						);			
	WX4A_CP1_Out	:	CpABS_Out;
	WX4A_CP2_CI		: 	CpABS_CI := (
//						//bHomeStart_PI:= , 
//						//Stop_PI:= , 
//						//Reset_VI:= , 
//						//JogExecute_VI:= , 
//						//JogSlow_VI:= , 
//						//CW_VI:= , 
//						PPRset_CI:= 2 , 
//						cntPulseSet_CI:= 32778 , //set for 1 degree per pulse
//						HomingSet_CI:= 3 ,
//						GearRatio_CI:= 3 , 
//						Lead_CI:= 8 , 
//						MechDriveType_CI:= 2, 
//						InputFilter_CI:= 7 , 
//						SWLimit_Hi_CI:= 180 , 
//						SWLimit_Lo_CI:= -90, 
//						Limit_NC_NO_CI:= 1, 	//add sensor if more protection needed
//						ABSEncoderScaler_CI := 131,		//converts 1 cp pulse to encoder counts (scale and adjust this and cntPulseSet_CI to scale to imperial or metric)
//						ABSEncoderZero_CI := 2089769026 , //will need to change if 'cntPulseSet_CI' is changed or the tolerance will need to be checked to see how close to limit
//						ABSHiLimit_CI	:= 2089792841, //will need to change if 'cntPulseSet_CI' is changed or the tolerance will need to be checked to see how close to limit
//						ABSLoLimit_CI := 2089757112 //will need to change if 'cntPulseSet_CI' is changed or the tolerance will need to be checked to see how close to limit
//						//abs currently set for -90 deg to 180 deg
//						,
//						DisPerPulse_CI :=1,
//						MoveABSTol_CI :=1.5
						);			
	WX4A_CP2_Out	:	CpABS_Out;
	WX4A_CP3_CI		: 	CpABS_CI := (
//						//bHomeStart_PI:= , 
//						//Stop_PI:= , 
//						//Reset_VI:= , 
//						//JogExecute_VI:= , 
//						//JogSlow_VI:= , 
//						//CW_VI:= , 
//						PPRset_CI:= 2 , 
//						cntPulseSet_CI:= 800 , 
//						HomingSet_CI:= 2 ,
//						GearRatio_CI:= 3 , 
//						Lead_CI:= 8 , 
//						MechDriveType_CI:= 2, 
//						InputFilter_CI:= 7 , 
//						SWLimit_Hi_CI:= 100 , 
//						SWLimit_Lo_CI:= -125, 
//						Limit_NC_NO_CI:= 1,
//						DisPerPulse_CI :=1,
//						MoveABSTol_CI :=1.5
						
						);			
	WX4A_CP3_Out	:	CpABS_Out;
	WX4B_CP1_CI		: 	CpABS_CI := (
//						//bHomeStart_PI:= , 
//						//Stop_PI:= , 
//						//Reset_VI:= , 
//						//JogExecute_VI:= , 
//						//JogSlow_VI:= , 
//						//CW_VI:= , 
//						PPRset_CI:= 2 , 
//						cntPulseSet_CI:= 32000 , 
//						HomingSet_CI:= 3 ,
//						GearRatio_CI:= 3 , 
//						Lead_CI:= 8 , 
//						MechDriveType_CI:= 2, 
//						InputFilter_CI:= 7 , 
//						SWLimit_Hi_CI:= 150 , 
//						SWLimit_Lo_CI:= 0, 
//						Limit_NC_NO_CI:= 0, 
//						ABSEncoderScaler_CI := -950,		//converts 1 cp pulse to encoder counts (scale and adjust this and cntPulseSet_CI to scale to imperial or metric)
//						ABSEncoderZero_CI := 2117612704 , //will need to change if 'cntPulseSet_CI' is changed or the tolerance will need to be checked to see how close to limit
//						ABSHiLimit_CI	:= 2117613849, //will need to change if 'cntPulseSet_CI' is changed or the tolerance will need to be checked to see how close to limit
//						ABSLoLimit_CI := 2117469332 //will need to change if 'cntPulseSet_CI' is changed or the tolerance will need to be checked to see how close to limit
//						//swap ABS Hi and ABS Lo if encoder is mounted opposite.
//						,
//						DisPerPulse_CI :=1,
//						MoveABSTol_CI :=1.5
						);			
	WX4B_CP1_Out	:	CpABS_Out;
	WX4B_CP2_CI		: 	CpABS_CI := (
//						//bHomeStart_PI:= , 
//						//Stop_PI:= , 
//						//Reset_VI:= , 
//						//JogExecute_VI:= , 
//						//JogSlow_VI:= , 
//						//CW_VI:= , 
//						PPRset_CI:= 2 , 
//						cntPulseSet_CI:= 32778 , //set for 1 degree per pulse
//						HomingSet_CI:= 3 ,
//						GearRatio_CI:= 3 , 
//						Lead_CI:= 8 , 
//						MechDriveType_CI:= 2, 
//						InputFilter_CI:= 7 , 
//						SWLimit_Hi_CI:= 180 , 
//						SWLimit_Lo_CI:= -90, 
//						Limit_NC_NO_CI:= 1, 	//add sensor if more protection needed later
//						ABSEncoderScaler_CI := 132,		//converts 1 cp pulse to encoder counts (scale and adjust this and cntPulseSet_CI to scale to imperial or metric)
//						ABSEncoderZero_CI := 2117532059	 , //will need to change if 'cntPulseSet_CI' is changed or the tolerance will need to be checked to see how close to limit
//						ABSHiLimit_CI	:= 2117555547, //will need to change if 'cntPulseSet_CI' is changed or the tolerance will need to be checked to see how close to limit
//						ABSLoLimit_CI := 2117520354 //will need to change if 'cntPulseSet_CI' is changed or the tolerance will need to be checked to see how close to limit
//						//abs currently set for -90 deg to 180 deg
//						,
//						DisPerPulse_CI :=1,
//						MoveABSTol_CI :=1.5
						);
	WX4B_CP2_Out	:	CpABS_Out;
	
	WX4B_CP3_CI		: 	CpABS_CI := ( //not config yet
//						//bHomeStart_PI:= , 
//						//Stop_PI:= , 
//						//Reset_VI:= , 
//						//JogExecute_VI:= , 
//						//JogSlow_VI:= , 
//						//CW_VI:= , 
//						PPRset_CI:= 2 , 
//						cntPulseSet_CI:= 800 , 
//						HomingSet_CI:= 2 ,
//						GearRatio_CI:= 3 , 
//						Lead_CI:= 8 , 
//						MechDriveType_CI:= 2, 
//						InputFilter_CI:= 7 , 
//						SWLimit_Hi_CI:= 150 , 
//						SWLimit_Lo_CI:= 0, 
//						Limit_NC_NO_CI:= 1,
//						DisPerPulse_CI :=1,
//						MoveABSTol_CI :=1.5
						
						
						);			
	WX4B_CP3_Out	:	CpABS_Out;
						
END_VAR

// ---- Machine System/GVLs/GVL_Job.TcGVL
{attribute 'qualified_only'}
VAR_GLOBAL
	FinishedWithSprayZoneSD1 : BOOL;
	FinishedWithSprayZoneSD2 : BOOL;
	
END_VAR

// ---- Machine System/GVLs/GVL_Log.TcGVL
{attribute 'qualified_only'}
VAR_GLOBAL
	NewMeasure : BOOL;
	PointLogged : BOOL;
	ReadytoLog 	: BOOL := TRUE;
	
	XCur		: STRING;
	YCur		: STRING;
	ZCur		: STRING;
	RCur		: STRING;
	VCur		: STRING;
	Dist		: STRING;
	
	XRef		: STRING;
	YRef		: STRING;
	ZRef		: STRING;
	RRef		: STRING;
	VRef		: STRING;
	DistRef		: STRING;
	
	
END_VAR

// ---- Machine System/GVLs/GVL_SAF.TcGVL
{attribute 'qualified_only'}
VAR_GLOBAL
	Estop1a 		AT %Q* : BOOL;
	Estop1b 		AT %Q* : BOOL;
	ErrorAcknowledgment AT %Q* : BOOL;
	Run 			AT %Q* : BOOL;
	InRun			AT %I* : BOOL;
	ComErr			AT %I* : BOOL;
	FbErr			AT %I* : BOOL;
	EStopReset 		AT %Q* : BOOL;
	EStopMCR 		AT %I* : BOOL;
	EStopError 		AT %I* : BOOL;	//error from main estop safety fb block
	EStopError1		AT %I* : BOOL;	//error from c4 estop safety fb block (same safe inputs as main estop)
	EstopError2 	AT %I* : BOOL;	//error from c5 estop safety fb block (same safe inputs as main estop)
	WX_On 			AT %Q* : BOOL;	//plc variable to drive safety outputs for c4 and c5 contactors (wx boxes)
	EDM_Error_C4 	AT %I* : BOOL;
	EDM_Error_C5 	AT %I* : BOOL;
	EStopOK			AT %I* : BOOL;
	DeadmanEnable	AT %I* : BOOL;  //from C3:SI1
	
	//plc flag
	SafetyOk		AT %I* : BOOL;
END_VAR

// ---- Machine System/GVLs/GVL_IO.TcGVL
VAR_GLOBAL
	//Digital Inputs
	bEstopPB AT %I* : BOOL; 
	iFeedrateOverridePot AT %I* : INT := 32767;
	iSpindleOverridePot AT %I* : INT := 32767;
	iSpindleLoad AT %I* : INT;
	//home and limit sensors
	bXHomeSwitch AT %I* : BOOL;
	bYHomeSwitch AT %I* : BOOL;
	bZHomeSwitch AT %I* : BOOL;
	bAHomeSwitch AT %I* : BOOL;
	bCHomeSwitch AT %I* : BOOL;
	bHi_A AT %I* : BOOL;
	bLo_A AT %I* : BOOL;
	bHi_C AT %I* : BOOL;
	bLo_C AT %I* : BOOL;
	
	// Temperature Analog
	Thermocouple AT %I*: REAL := 0; // C3 EL3024 Channel 3 analog 4-20mA from thermocouple range 0-32767
	rAIInput1 : REAL;
	rAIInput2 : REAL;
	rAIInput3 : REAL;
	
	//Distance Analog
	iDistSens	AT %I*	: INT;	//analog distance sensor on z axis to measure tool
	
	//trunnion sensors
	bTrunCW AT %I* : BOOL;
	bTrunCCW AT %I* : BOOL;
	bTrun0 AT %I* : BOOL;
	bTrunOver AT %I* : BOOL;
	bTrunClampOn : BOOL :=true; // Trunnion clamp
	bTrunClampOnLast : BOOL :=TRUE; //Track state of clamp to disallow change while estop or enable off
	bTrunClampEn : BOOL;
	
	iTrunSig AT %Q*: INT;
	//Trunion Clearpath rotary
	//bEnable 	AT 	%Q* 	: BOOL;		//found in cprot function
	bEnableCom	AT 	%I* 	: BOOL;
	bAcom		AT	%I* 	: BOOL;
	//bAout		AT 	%Q*		: BOOL;		//found in cprot function
	bBcom		AT	%I* 	: BOOL;
	//bBout		AT 	%Q*		: BOOL;		//found in cprot function
	bHLFBcom	AT	%I* 	: BOOL;		//red wire
	bHLFB24V	AT 	%Q*		: BOOL; 	//green wire
	
	// gun valves
	bAceOn AT %Q* : BOOL;	// acetone gun mac valve
	bSprayOn AT %Q* : BOOL; // spray gun mac valve
	// smc valve outputs - one must be true and one must be false (a true b false or A false B true)
	bVa1A AT %Q* :BOOL;
	bVa1B AT %Q* :BOOL;
	bVa2A AT %Q* :BOOL;
	bVa2B AT %Q* :BOOL;
	bVa3A AT %Q* :BOOL;
	bVa3B AT %Q* :BOOL;
	bva4A AT %Q* : BOOL;
	bVa4B AT %Q* :BOOL;
	bVa5A AT %Q* :BOOL;
	bVa5B AT %Q* :BOOL;
	bVa6A AT %Q* :BOOL;
	bVa6B AT %Q* :BOOL;
	bVa7A AT %Q* :BOOL;
	bVa7B AT %Q* :BOOL;
	bVa8A AT %Q* :BOOL;
	bVa8B AT %Q* :BOOL;
	bVa9A AT %Q* :BOOL;
	bVa9B AT %Q* :BOOL;
	bVa10A AT %Q* :BOOL;
	bVa10B AT %Q* :BOOL;
	bVa11A AT %Q* :BOOL;
	bVa11B AT %Q* :BOOL;
	bVa12A AT %Q* :BOOL;
	bVa12B AT %Q* :BOOL;
	bVa13A AT %Q* :BOOL;	
	bVa13B AT %Q* :BOOL;
	bVa14A AT %Q* :BOOL;
	bVa14B AT %Q* :BOOL;
	bVa15A AT %Q* :BOOL;
	bVa15B AT %Q* :BOOL;
	bVa16A AT %Q* :BOOL;
	bVa16B AT %Q* :BOOL;
	
	WX1 : sBogie;
	WX2 : sBogie;
	WX3 : sBogie;
	WX4 : sBogie;
	
	//C6
	KM1_ContactorOn  AT %Q* : BOOL;
	KM2_ContactorOn  AT %Q* : BOOL;
	//C3
	FilterManometer AT %I*: INT; // Air Filter Elements differential pressure sensor
	gasSensor AT %I* : INT; // Styrene level sensor
	
END_VAR

// ---- Machine System/GVLs/GVL_Machine.TcGVL
VAR_GLOBAL
	pX: POINTER TO HIGH_LEVEL_INTERFACE_AX;
	pY: POINTER TO HIGH_LEVEL_INTERFACE_AX;
	pZ: POINTER TO HIGH_LEVEL_INTERFACE_AX;
	pCh0: POINTER TO HIGH_LEVEL_INTERFACE_CH;
	rX_ActPos : LREAL;
	rY_ActPos : LREAL;
	rZ_ActPos : LREAL;
	bAllAxisOkToEnable 	: BOOL;	
	bPLC_ForceEstop 	: BOOL;
	nCommandedRPM		: DINT;
	stVirtualHBA		: ARRAY[0..1] OF ST_CNCVirtualHBA;
	HeaterOnRequest		: LREAL;
	fSetpointValueToScope: LREAL;
	fActualValueToScope	 : LREAL;
	fOutToScope			: LREAL;
	fPIDLoop1ControlValue : LREAL;
	fPIDLoop1ProcessValue : LREAL;
	HeatOnRequest : BOOL;
	
END_VAR

VAR_GLOBAL CONSTANT
	MAX_CSV_ROWS 			: UDINT := 250;
	MAX_CSV_COLUMNS 		: UDINT := 1;
	MAX_CSV_FIELD_LENGTH	: UDINT := 100;
END_VAR

// ---- Machine System/PRGs/PID/PRG_PID_CALL.TcPOU
PROGRAM PRG_PID_CALL
VAR
	
END_VAR




// C3 EL3024 Channel 3 analog 4-20mA from thermocouple range 0-32767
// Measure -40F to 140F
GVL_IO.rAIInput3 := (Thermocouple/(32767.0 - 0.0))* 100;

HeaterOnRequest := PRG_FB_CTRL_PID.fOut;
PRG_FB_CTRL_PID();

//Call simulated PID for debugging locally. Comment out after commissioning
//PRG_SIM_PROCESS();

END_PROGRAM

// ---- Machine System/PRGs/PID/PRG_FB_CTRL_PID.TcPOU
PROGRAM PRG_FB_CTRL_PID
VAR
	fSetpointValue					: LREAL		:= 85.0;
	fActualValue					: LREAL;
	fManSyncValue					: LREAL;
	bSync							: BOOL;

	fOut							: LREAL;
	
	bHold							: BOOL;

	eMode							: E_CTRL_MODE;
	stCTRL_PID_PARAMS				: ST_CTRL_PID_PARAMS;

	eErrorId						: E_CTRL_ERRORCODES;
	bError							: BOOL;
	bARWactive						: BOOL;

	(* controller *)
	fbCTRL_PID						: FB_CTRL_PID;

	bInit							: BOOL	:= TRUE;
	fbTON							: TON;
	TcHmiToggleButtonHeaterOnOff    : BOOL;
END_VAR


	

IF bInit THEN
	(* init parameter struct *)
	stCTRL_PID_PARAMS.tCtrlCycleTime		:= T#500MS;
	stCTRL_PID_PARAMS.tTaskCycleTime		:= T#100MS;
	stCTRL_PID_PARAMS.fKp					:= 3.0;			(* proportional gain Kp				*)
	stCTRL_PID_PARAMS.tTn					:= T#20S;		(*  Tn								*)
	stCTRL_PID_PARAMS.tTv					:= T#200MS;		(*  Tv								*)
	stCTRL_PID_PARAMS.tTd					:= T#100MS;		(*  Td								*)
	stCTRL_PID_PARAMS.fOutMaxLimit			:=  100;		(* maximum output limit				*)
	stCTRL_PID_PARAMS.fOutMinLimit			:=  0.0;		(* minimum output limit				*)

	(* set the mode to ACTIVE --> normal operation *)
	eMode := eCTRL_MODE_ACTIVE;

	(* reset the init flag *)
	bInit := FALSE;
END_IF

(*TYPE E_CTRL_MODE :
(
    eCTRL_MODE_IDLE     := 0, 
    eCTRL_MODE_PASSIVE     := 1, 
    eCTRL_MODE_ACTIVE     := 2, 
    eCTRL_MODE_RESET     := 3, 
    eCTRL_MODE_MANUAL     := 4, 
    eCTRL_MODE_TUNE     := 5, 
    eCTRL_MODE_SELFTEST    := 6, 
    eCTRL_MODE_SYNC_MOVEMENT := 7 
)
END_TYPE*)

fActualValue := GVL_IO.rAIInput3; //Get process variable Temperature from analog input C3, AI1 Channel 3 value

(* copy var to scope var *)
GVL_Machine.fSetpointValueToScope 	:= fSetpointValue;
GVL_Machine.fActualValueToScope 	:= fActualValue;
GVL_Machine.fOutToScope 			:= fOut;

(* call controller *)
fbCTRL_PID(		fSetpointValue		:= fSetpointValue,
				fActualValue		:= fActualValue,
				fManSyncValue		:= fOut,
				bSync				:= bSync,
				eMode				:= eMode,
				bHold				:= bHold,
				stParams			:= stCTRL_PID_PARAMS,
				fOut				=> fOut,
				bARWactive			=> bARWactive,
				eErrorId			=> eErrorId,
				bError				=> bError
				);

(*IF eMode = 	eCTRL_MODE_ACTIVE THEN // Bumpless switch logic for switching PID for Manual to Automatic. The setpoint value needs TO follow the process value feedback
	fOut := fOut;		
END_IF				

IF eMode = 	eCTRL_MODE_ACTIVE THEN // Bumpless switch logic for switching PID for Automatic to Manual. The setpoint value needs to follow the process value feedback
	fSetpointValue := fActualValue;		
END_IF	*)

IF 	GVL_Machine.fOutToScope >= 10 OR TcHmiToggleButtonHeaterOnOff THEN
	 GVL_Machine.HeatOnRequest := TRUE;
	ELSE
	 GVL_Machine.HeatOnRequest := FALSE;
END_IF

END_PROGRAM

// ---- FAST.TcPOU
PROGRAM FAST
VAR
	nChan : INT;
	MOS_TS: INT;
END_VAR

(****************************************************************************************)
(*	  							Wait for HLI initialization								*)
(****************************************************************************************)
IF NOT CNCSystem.bHLIInit THEN
	RETURN;
END_IF

(* Programm call for MOS_TS M functions *)
// PRG_FastMFunctions();

END_PROGRAM

// ---- MAIN.TcPOU
PROGRAM MAIN
VAR
  
END_VAR



// everything related to time
	P_Timer();
	
	
// EventLogger
	P_EventLogger();

FirstScan();
// temporarily disabled by Kirk 
HLI3_Init(); 

//PRG_Sequence();
(* Call CNC related code only if the HLI has been initialized succesfully! *)
 IF CNCSystem.bHLIInit THEN
	PRG_CNCAxesHandler();    	
	PRG_CNCManualMode();
	PRG_CNCChannelHandler();	
	PRG_CNCVariablesViewer();
	PRG_ManualFnc();	
	myPRG_AxisHomeSwitches_1();
	myVE_Vars(); //call this before MCodes just to be sure data was pulled and updated for each potential MCODE Call [Add a buffer to mcode rtrig if ve does not compute from same gcode line call ie[ve.wxv=90 M510]
	myM_CODES();
////	myPressure();
//	myGun();
//	myCounter();
	mySafety();
	SafetyConnect();
	ModeHandle();
	//myHMIPLCRECIPE();
	//myDistance();
	WX_CP();
	WX_CP_Simple();
	Bogie();
	//myCNC_Call_Spray();
	CNC_HMI_HLI_Added_Code(); //display for new hmi variables
	BogieSettings();
	RollerDoors();
	PersonnelDoor();
	Heraus_Heater_Control();
	
//	 		(* Conveyor Programs *)
	
	Input_Buffering();
	MOTOR_FAULTS();
	JAM_FAULTS();
	OUTPUTS();
	//Ventilation();
	GL1_Transfer_Traverse();
	GL10_Transfer_Traverse();
	GL11_Transfer();
	GL2_Transfer();
	GL3_Accumulation();
	GL4_Accumulation();
	GL5A_Accumulation();
	GL5B_Accumulation();
	GL6_Conveyor();
	GL7_Conveyor();
	GL8_Conveyor();
	GL9_Conveyor();

			(* Rib Machine Programs *)
	Guarding_Safety();
	Input_Buffering_RB();
	START_STOP();
	Index_and_measure();
	Fault_Logic();
	Lift_Raise_and_Lower();
	Clamp_and_cut();
	Interlocks_to_Main_Line();
	// Outputs_RB();
	
END_IF
(* Reset the reset flag from HMI *)
PLCReset := FALSE;

END_PROGRAM

// ---- Machine System/PRGs/ALARM AND STATUS/P_Timer.TcPOU
PROGRAM P_Timer 
VAR
	fbSystemTime 		: FB_LocalSystemTime;
	dtCurrentDateTime 	: DT;
	sCurrentDateTime 	: STRING;
	sDateTime			: STRING;		
	bSecond				: BOOL;
	nSecond 			: WORD;
	bPulsels			: BOOL;
	
	fbRtSecond 			: R_TRIG;
	fbLow_ls			: TON;
	fbHigh_ls 			: TOF;
END_VAR

// synchronize system time 
	fbSystemTime(
		bEnable		:= TRUE, 
		dwCycle		:= 5, 
		dwOpt		:= 1
	);

	dtCurrentDateTime	:= SYSTEMTIME_TO_DT(fbSystemTime.systemTime); 
	sCurrentDateTime	:= MID(DT_TO_STRING(dtCurrentDateTime), 19, 4);

// convert timestamp because ':' invalid in file name 
	sDateTime := sCurrentDateTime; 
	sDateTime := replace (sDateTime,'-', 1, 11); 
	sDateTime := replace (sDateTime,'-', 1, 14); 
	sDateTime := replace (sDateTime,'-', 1, 17);
	
// 1 sec. trigger
	fbRtSecond (CLK 	:= fbSystemTime.systemTime.wSecond <> nSecond, Q => bSecond);
 	nSecond				:= fbSystemTime.systemTime.wSecond;
	
// 1 sec. blinking puls
	fbLow_ls(IN 		:= NOT bPulsels, PT:= T#500MS);
	fbHigh_ls(IN		:= fbLow_ls.Q,   PT:= T#500MS, Q => bPulsels);

END_PROGRAM

// ---- Machine System/PRGs/ALARM AND STATUS/P_EventLogger.TcPOU
PROGRAM P_EventLogger
VAR
	fbEventlogger		: FB_TcEventlogger;
	bClearAlarms		: BOOL;
	bConfirmAlarms 		: BOOL; 
	bClearLoggedEvents 	: BOOL; 
	bExportLoggedEvents : BOOL; 
	fbRtExport			: R_TRIG; 
	fbCsvExportSetting  : FB_TcEventCsvExportSettings; 
	fbExportFilter 		: FB_TcEventFilter; 
	sExportFileName 	: STRING := 'C:\temp\Eventlogger-export.csv';
	
	fbEventAlarm		: ARRAY[0..500] OF FB_EventAlarm;
	aClass1Alarm		: ARRAY[0..500] OF BOOL;	
	aClass2Alarm		: ARRAY[0..500] OF BOOL;	
	aClass3Alarm		: ARRAY[0..500] OF BOOL;	
	fbEventWarning 		: ARRAY[0..500] OF FB_EventMessage;
	aWarning			: ARRAY[0..512] OF BOOL;
	fbEventInfo 		: ARRAY[0..500] OF FB_EventMessage;
	aInfo				: ARRAY[0..500] OF BOOL;
  
	hr					: HRESULT;
	hrLastError 		: HRESULT;
	
END_VAR

Event_Calls(); 				// Program to turn Alarms on
a_010_AlarmsClass1(); 		// alarms class 1, emergency stop, safety doors, power supply, etc.
a_010_AlarmsClass2(); 		// alarms class 2, movements, drives, pneumatic cylinder, etc.
a_010_AlarmsClass3(); 		// alarms class 3, process, level, temperature, conductivity, etc.

a_020_Warnings(); 			// warnings, filter change, refilling of tanks, pre-alarms, etc.

a_030_Infos(); 				// messages, audit-trail, etc.

a_040_ConfirmLoggedAlarms();// confirm all logged alarms

(*a_050_ClearLoggedAlarms ();// clear all logged events PLC*)

a_060_ClearLoggedEvents(); // clear all logged events PLC

a_070_ExportLoggedEvents();// export logged events csv file

ACTION a_010_AlarmsClass1:

//Alarms Class 1 
	fbEventAlarm[0](
		bEvent			:=	aClass1Alarm[0],
		nEventID		:=	4096,
		sSource			:=	'TwinSAFE Program'
	);
	fbEventAlarm[1](
		bEvent			:=	aClass1Alarm[1],
		nEventID		:=	4097,
		sSource			:=	'GL1 Motor Fault'
	);
	fbEventAlarm[2](
		bEvent			:=	aClass1Alarm[2],
		nEventID		:=	4098,
		sSource			:=	'GL2 Motor Fault'
	);
	fbEventAlarm[3](
		bEvent			:=	aClass1Alarm[3],
		nEventID		:=	4099,
		sSource			:=	'GL3 Motor Fault'
	);
	fbEventAlarm[4](
		bEvent			:=	aClass1Alarm[4],
		nEventID		:=	4100,
		sSource			:=	'GL4 Motor Fault'
	);
	fbEventAlarm[5](
		bEvent			:=	aClass1Alarm[5],
		nEventID		:=	4101,
		sSource			:=	'GL5A Motor Fault'
	);
	fbEventAlarm[6](
		bEvent			:=	aClass1Alarm[6],
		nEventID		:=	4102,
		sSource			:=	'GL5B Motor Fault'
	);
	fbEventAlarm[7](
		bEvent			:=	aClass1Alarm[7],
		nEventID		:=	4103,
		sSource			:=	'GL6 Motor Fault'
	);
	fbEventAlarm[8](
		bEvent			:=	aClass1Alarm[8],
		nEventID		:=	4104,
		sSource			:=	'GL7 Motor Fault'
	);
	fbEventAlarm[9](
		bEvent			:=	aClass1Alarm[9],
		nEventID		:=	4105,
		sSource			:=	'GL8 Motor Fault'
	);
	fbEventAlarm[10](
		bEvent			:=	aClass1Alarm[10],
		nEventID		:=	4106,
		sSource			:=	'GL9 Motor Fault'
	);
	fbEventAlarm[11](
		bEvent			:=	aClass1Alarm[11],
		nEventID		:=	4107,
		sSource			:=	'GL10 Motor Fault'
	);
	fbEventAlarm[12](
		bEvent			:=	aClass1Alarm[12],
		nEventID		:=	4108,
		sSource			:=	'GL11 Motor Fault'
	);
	fbEventAlarm[13](
		bEvent			:=	aClass1Alarm[13],
		nEventID		:=	4109,
		sSource			:=	'GL12 Motor Fault'
	);
END_ACTION

ACTION a_010_AlarmsClass2:
//Alarms Class 2 
	fbEventAlarm[14](
		bEvent			:=	aClass2Alarm[0],
		nEventID		:=	8192,
		sSource			:=	'GL1 jam'
	);
	fbEventAlarm[15](
		bEvent			:=	aClass2Alarm[1],
		nEventID		:=	8193,
		sSource			:=	'GL2 jam'
	);
	fbEventAlarm[16](
		bEvent			:=	aClass2Alarm[2],
		nEventID		:=	8194,
		sSource			:=	'GL3 jam'
	);
	fbEventAlarm[17](
		bEvent			:=	aClass2Alarm[3],
		nEventID		:=	8195,
		sSource			:=	'GL4 jam'
	);
	fbEventAlarm[18](
		bEvent			:=	aClass2Alarm[4],
		nEventID		:=	8196,
		sSource			:=	'GL5A jam'
	);
	fbEventAlarm[19](
		bEvent			:=	aClass2Alarm[5],
		nEventID		:=	8197,
		sSource			:=	'GL5B jam'
	);
	fbEventAlarm[20](
		bEvent			:=	aClass2Alarm[6],
		nEventID		:=	8198,
		sSource			:=	'GL6 jam'
	);
	fbEventAlarm[21](
		bEvent			:=	aClass2Alarm[7],
		nEventID		:=	8199,
		sSource			:=	'GL7 jam'
	);
	fbEventAlarm[22](
		bEvent			:=	aClass2Alarm[8],
		nEventID		:=	8200,
		sSource			:=	'GL8 jam'
	);
	fbEventAlarm[23](
		bEvent			:=	aClass2Alarm[9],
		nEventID		:=	8201,
		sSource			:=	'GL9 jam'
	);
	fbEventAlarm[24](
		bEvent			:=	aClass2Alarm[10],
		nEventID		:=	8202,
		sSource			:=	'GL10 jam'
	);
	fbEventAlarm[25](
		bEvent			:=	aClass2Alarm[11],
		nEventID		:=	8203,
		sSource			:=	'GL11 jam'
	);
	fbEventAlarm[26](
		bEvent			:=	aClass2Alarm[12],
		nEventID		:=	8204,
		sSource			:=	'GL12 jam'
	);
END_ACTION

ACTION a_010_AlarmsClass3:
//Alarms Class 3 
	fbEventAlarm[30](
		bEvent			:=	aClass3Alarm[0],
		nEventID		:=	4116,
		sSource			:=	'Air Filter'
	);
	fbEventAlarm[31](
		bEvent			:=	aClass3Alarm[1],
		nEventID		:=	4117,
		sSource			:=	'Air Filter'
	);
	fbEventAlarm[32](
		bEvent			:=	aClass3Alarm[2],
		nEventID		:=	4118,
		sSource			:=	'Styrene'
	);
	fbEventAlarm[33](
		bEvent			:=	aClass3Alarm[3],
		nEventID		:=	4119,
		sSource			:=	'Class3Alarm 3'
	);
	fbEventAlarm[34](
		bEvent			:=	aClass3Alarm[4],
		nEventID		:=	4120,
		sSource			:=	'Class3Alarm 4'
	);
	fbEventAlarm[35](
		bEvent			:=	aClass3Alarm[5],
		nEventID		:=	4121,
		sSource			:=	'Class3Alarm 5'
	);
	fbEventAlarm[36](
		bEvent			:=	aClass3Alarm[6],
		nEventID		:=	4122,
		sSource			:=	'Class3Alarm 6'
	);
	fbEventAlarm[37](
		bEvent			:=	aClass3Alarm[7],
		nEventID		:=	4123,
		sSource			:=	'Class3Alarm 7'
	);
	fbEventAlarm[38](
		bEvent			:=	aClass3Alarm[8],
		nEventID		:=	4124,
		sSource			:=	'Class3Alarm 8'
	);
	fbEventAlarm[39](
		bEvent			:=	aClass3Alarm[9],
		nEventID		:=	4125,
		sSource			:=	'Class3Alarm 9'
	);
END_ACTION

ACTION a_020_Warnings:
// Warning 
	fbEventWarning[0](
		bEvent 		:= 	aWarning[0],
		nEventID	:=	1280,
		sSource		:=	'Styrene Level'
	);
	fbEventWarning[1](
		bEvent 		:= 	aWarning[1],
		nEventID	:=	1281,
		sSource		:=	'Roll Door 1'
	);
	fbEventWarning[2](
		bEvent 		:= 	aWarning[2],
		nEventID	:=	1282,
		sSource		:=	'Roll Door 2'
	);
	fbEventWarning[3](
		bEvent 		:= 	aWarning[3],
		nEventID	:=	1283,
		sSource		:=	'Roll Door 3'
	);
	fbEventWarning[4](
		bEvent 		:= 	aWarning[4],
		nEventID	:=	1284,
		sSource		:=	'Warning 4'
	);
	fbEventWarning[5](
		bEvent 		:= 	aWarning[5],
		nEventID	:=	1285,
		sSource		:=	'Warning 5'
	);
	fbEventWarning[6](
		bEvent 		:= 	aWarning[6],
		nEventID	:=	1286,
		sSource		:=	'Warning 6'
	);
	fbEventWarning[7](
		bEvent 		:= 	aWarning[7],
		nEventID	:=	1287,
		sSource		:=	'Warning 7'
	);
	fbEventWarning[8](
		bEvent 		:= 	aWarning[8],
		nEventID	:=	1288,
		sSource		:=	'Warning 8'
	);
	fbEventWarning[9](
		bEvent 		:= 	aWarning[9],
		nEventID	:=	1289,
		sSource		:=	'Warning 9'
	);
	fbEventWarning[10](
		bEvent 		:= 	aWarning[10],
		nEventID	:=	1290,
		sSource		:=	'Warning 10'
	);
	fbEventWarning[11](
		bEvent 		:= 	aWarning[11],
		nEventID	:=	1291,
		sSource		:=	'Warning 11'
	);
	fbEventWarning[12](
		bEvent 		:= 	aWarning[12],
		nEventID	:=	1292,
		sSource		:=	'Warning 12'
	);
	fbEventWarning[13](
		bEvent 		:= 	aWarning[13],
		nEventID	:=	1293,
		sSource		:=	'Warning 13'
	);
	fbEventWarning[14](
		bEvent 		:= 	aWarning[14],
		nEventID	:=	1294,
		sSource		:=	'Warning 14'
	);
	fbEventWarning[15](
		bEvent 		:= 	aWarning[15],
		nEventID	:=	1295,
		sSource		:=	'Warning 15'
	);
	fbEventWarning[16](
		bEvent 		:= 	aWarning[16],
		nEventID	:=	1296,
		sSource		:=	'Warning 16'
	);
	fbEventWarning[17](
		bEvent 		:= 	aWarning[17],
		nEventID	:=	1297,
		sSource		:=	'Warning 17'
	);
	fbEventWarning[18](
		bEvent 		:= 	aWarning[18],
		nEventID	:=	1298,
		sSource		:=	'Warning 18'
	);
	fbEventWarning[19](
		bEvent 		:= 	aWarning[19],
		nEventID	:=	1299,
		sSource		:=	'Warning 19'
	);
END_ACTION

ACTION a_030_Infos:
// Info 
	fbEventInfo[0](
		bEvent 		:= 	aInfo[0],
		nEventID	:=	0,
		sSource		:=	'Info 0'
	);
	fbEventInfo[1](
		bEvent 		:= 	aInfo[1],
		nEventID	:=	1,
		sSource		:=	'Info 1'
	);
	fbEventInfo[2](
		bEvent 		:= 	aInfo[2],
		nEventID	:=	2,
		sSource		:=	'Info 2'
	);
	fbEventInfo[3](
		bEvent 		:= 	aInfo[3],
		nEventID	:=	3,
		sSource		:=	'Info 3'
	);
	fbEventInfo[4](
		bEvent 		:= 	aInfo[4],
		nEventID	:=	4,
		sSource		:=	'Info 4'
	);
	fbEventInfo[5](
		bEvent 		:= 	aInfo[5],
		nEventID	:=	5,
		sSource		:=	'Info 5'
	);
	fbEventInfo[6](
		bEvent 		:= 	aInfo[6],
		nEventID	:=	6,
		sSource		:=	'Info 6'
	);
	fbEventInfo[7](
		bEvent 		:= 	aInfo[7],
		nEventID	:=	7,
		sSource		:=	'Info 7'
	);
	fbEventInfo[8](
		bEvent 		:= 	aInfo[8],
		nEventID	:=	8,
		sSource		:=	'Info 8'
	);
	fbEventInfo[9](
		bEvent 		:= 	aInfo[9],
		nEventID	:=	9,
		sSource		:=	'Info 9'
	);
	fbEventInfo[10](
		bEvent 		:= 	aInfo[10],
		nEventID	:=	10,
		sSource		:=	'Info 10'
	);
	fbEventInfo[11](
		bEvent 		:= 	aInfo[11],
		nEventID	:=	11,
		sSource		:=	'Info 11'
	);
	fbEventInfo[12](
		bEvent 		:= 	aInfo[12],
		nEventID	:=	12,
		sSource		:=	'Info 12'
	);
	fbEventInfo[13](
		bEvent 		:= 	aInfo[13],
		nEventID	:=	13,
		sSource		:=	'Info 13'
	);
	fbEventInfo[14](
		bEvent 		:= 	aInfo[14],
		nEventID	:=	14,
		sSource		:=	'Info 14'
	);
	fbEventInfo[15](
		bEvent 		:= 	aInfo[15],
		nEventID	:=	15,
		sSource		:=	'Info 15'
	);
	fbEventInfo[16](
		bEvent 		:= 	aInfo[16],
		nEventID	:=	16,
		sSource		:=	'Info 16'
	);
	fbEventInfo[17](
		bEvent 		:= 	aInfo[17],
		nEventID	:=	17,
		sSource		:=	'Info 17'
	);
	fbEventInfo[18](
		bEvent 		:= 	aInfo[18],
		nEventID	:=	18,
		sSource		:=	'Info 18'
	);
	fbEventInfo[19](
		bEvent 		:= 	aInfo[19],
		nEventID	:=	19,
		sSource		:=	'Info 19'
	);
END_ACTION

ACTION a_040_ConfirmLoggedAlarms:
// confirmation of all alarms	

	IF bConfirmAlarms THEN
			hr:= fbEventLogger.ConfirmAllAlarms(0);
			IF FAILED(hr) THEN
				hrLastError := hr;
			END_IF
	END_IF
END_ACTION

ACTION a_050_ClearLoggedAlarms:
// reset ALL Alarms 
// must not be used!!! I reset the alarms in the corresponding instances

	(*IF bClearAlarms THEN
			hr := fbEventlogger.ClearAllAlarms(0,FALSE);
			IF FAILED(hr) THEN
					hrLastError := hr;
			END_IF
	END_IF*)
END_ACTION

ACTION a_060_ClearLoggedEvents:
// clear all logged events PLC Cache
	IF bClearLoggedEvents THEN
		bClearLoggedEvents := FALSE;
		fbEventlogger.ClearLoggedEvents(0);
	END_IF
END_ACTION

ACTION a_070_ExportLoggedEvents:
// create file name
	sExportFileName := CONCAT(CONCAT('C:\Temp\',P_Timer.sDateTime), '.csv');
	
// CSV export logged events. Without filter all logged events will be exported. 
// CSV file will be overvritten, an opened file fires an error
	fbRtExport (CLK:= bExportLoggedEvents); 
	IF bExportLoggedEvents THEN 
		IF fbRtExport.Q THEN
			fbCsvExportSetting.Clear(); 
			fbCsvExportSetting.AddLanguage(1031, 'German'); 
		//	fbCsvExportSetting. AddFilter (fbExportFilter);
		//	fbExportFilter.Clear().IsAlarm()AND_OP().EventClass.EqualTO (TC_EVENTS.myAlarmEventClass.x1000.uuidEventClass); 
		END_IF 
		IF fbEventLogger.ExportLoggedEvents(sExportFileName,fbCsvExportSetting, hrErrorCode=> hr) THEN
			bExportLoggedEvents:= FALSE; 
		END_IF 
	END_IF
END_ACTION

ACTION Event_Calls:


// alarms class 1, emergency stop, safety doors, power supply, etc.
	IF NOT gvl_saf.SafetyOk THEN aClass1Alarm[0] := 1; ELSE aClass1Alarm[0] := 0; END_IF
		
/////////////////////////// CONVEYOR MOTOR FAULTS
	
	
	IF GVL_Conveyors.GL1.Motor_Fault THEN aClass1Alarm[1] := 1; ELSE aClass1Alarm[1] := 0; END_IF // GL1 MOTOR FAULT
	
	IF GVL_Conveyors.GL2.Motor_Fault THEN aClass1Alarm[2] := 1; ELSE aClass1Alarm[2] := 0; END_IF // GL2 MOTOR FAULT
		
	IF GVL_Conveyors.GL3.Motor_Fault THEN aClass1Alarm[3] := 1; ELSE aClass1Alarm[3] := 0; END_IF // GL3 MOTOR FAULT
	
	IF GVL_Conveyors.GL4.Motor_Fault THEN aClass1Alarm[4] := 1; ELSE aClass1Alarm[4] := 0; END_IF // GL4 MOTOR FAULT
	
	IF GVL_Conveyors.GL5A.Motor_Fault THEN aClass1Alarm[5] := 1; ELSE aClass1Alarm[5] := 0; END_IF // GL5A MOTOR FAULT
	
	IF GVL_Conveyors.GL5B.Motor_Fault THEN aClass1Alarm[6] := 1; ELSE aClass1Alarm[5] := 0; END_IF // GL5B MOTOR FAULT
		
	IF GVL_Conveyors.GL6.Motor_Fault THEN aClass1Alarm[7] := 1; ELSE aClass1Alarm[7] := 0; END_IF // GL6 MOTOR FAULT
	
	IF GVL_Conveyors.GL7.Motor_Fault THEN aClass1Alarm[8] := 1; ELSE aClass1Alarm[8] := 0; END_IF // GL7 MOTOR FAULT
	
	IF GVL_Conveyors.GL8.Motor_Fault THEN aClass1Alarm[9] := 1; ELSE aClass1Alarm[9] := 0; END_IF // GL8 MOTOR FAULT
	
	IF GVL_Conveyors.GL9.Motor_Fault THEN aClass1Alarm[10] := 1; ELSE aClass1Alarm[10] := 0; END_IF // GL9 MOTOR FAULT
		
	IF GVL_Conveyors.GL10.Motor_Fault THEN aClass1Alarm[11] := 1; ELSE aClass1Alarm[11] := 0; END_IF // GL10 MOTOR FAULT
	
	IF GVL_Conveyors.GL11.Motor_Fault THEN aClass1Alarm[12] := 1; ELSE aClass1Alarm[12] := 0; END_IF // GL11 MOTOR FAULT
	
	IF GVL_Conveyors.GL12.Motor_Fault THEN aClass1Alarm[13] := 1; ELSE aClass1Alarm[13] := 0; END_IF // GL12 MOTOR FAULT
	
	
	//////////////////////////////CONVEYOR JAM FAULTS
	// alarms class 2, movements, drives, pneumatic cylinder, etc.
	
	IF GVL_Conveyors.GL1.Jam_Fault 	THEN aClass2Alarm[0] := 1; ELSE aClass2Alarm[0] := 0; END_IF // GL1 JAM FAULT
		
	IF GVL_Conveyors.GL2.Jam_Fault 	THEN aClass2Alarm[1] := 1; ELSE aClass2Alarm[1] := 0; END_IF // GL2 JAM FAULT
	
	IF GVL_Conveyors.GL3.Jam_Fault 	THEN aClass2Alarm[2] := 1; ELSE aClass2Alarm[2] := 0; END_IF // GL3 JAM FAULT
	
	IF GVL_Conveyors.GL4.Jam_Fault 	THEN aClass2Alarm[3] := 1; ELSE aClass2Alarm[3] := 0; END_IF // GL4 JAM FAULT
	
	IF GVL_Conveyors.GL5A.Jam_Fault	THEN aClass2Alarm[4] := 1; ELSE aClass2Alarm[4] := 0; END_IF // GL5A JAM FAULT

	IF GVL_Conveyors.GL5B.Jam_Fault	THEN aClass2Alarm[5] := 1; ELSE aClass2Alarm[5] := 0; END_IF // GL5B JAM FAULT
		
	IF GVL_Conveyors.GL6.Jam_Fault	THEN aClass2Alarm[6] := 1; ELSE aClass2Alarm[6] := 0; END_IF // GL6 JAM FAULT

	IF GVL_Conveyors.GL7.Jam_Fault	THEN aClass2Alarm[7] := 1; ELSE aClass2Alarm[7] := 0; END_IF // GL7 JAM FAULT
		
	IF GVL_Conveyors.GL8.Jam_Fault	THEN aClass2Alarm[8] := 1; ELSE aClass2Alarm[8] := 0; END_IF // GL8 JAM FAULT
		
	IF GVL_Conveyors.GL9.Jam_Fault	THEN aClass2Alarm[9] := 1; ELSE aClass2Alarm[9] := 0; END_IF // GL9 JAM FAULT
	
	IF GVL_Conveyors.GL10.Jam_Fault	THEN aClass2Alarm[10] := 1; ELSE aClass2Alarm[10] := 0; END_IF // GL10 JAM FAULT
		
	IF GVL_Conveyors.GL11.Jam_Fault	THEN aClass2Alarm[11] := 1; ELSE aClass2Alarm[11] := 0; END_IF // GL11 JAM FAULT
	
	IF GVL_Conveyors.GL12.Jam_Fault	THEN aClass2Alarm[12] := 1; ELSE aClass2Alarm[12] := 0; END_IF // GL12 JAM FAULT
	
	

// alarms class 3, process, level, temperature, conductivity, etc.

	IF Ventilation.FILTER_CHANGE_NEEDED		THEN aClass3Alarm[0] := 1; ELSE aClass3Alarm[0] := 0; END_IF
	
	IF Ventilation.FILTER_OBSTRUCTED_FAULT THEN aClass3Alarm[1] := 1; ELSE aClass3Alarm[1] := 0; END_IF
		
	IF Ventilation.gasSensorFaulted		THEN aClass3Alarm[2] := 1; ELSE aClass3Alarm[2] := 0; END_IF
	
		
	//IF NewBatch.ResinTote.ActualScaleWeight < NewBatch.ResinTote.EmptyScaleWeight
	//									THEN aClass3Alarm[2] := 1; ELSE aClass3Alarm[2] := 0; END_IF
		
	//IF GVL.FiltersNeedChangeOutMain		THEN aClass3Alarm[3] := 1; ELSE aClass3Alarm[3] := 0; END_IF
		
	//IF GVL.FiltersNeedChangeOutSpecial	THEN aClass3Alarm[4] := 1; ELSE aClass3Alarm[4] := 0; END_IF
		
	//IF NewBatch.MixerCaseStep = 900		THEN aClass3Alarm[5] := 1; ELSE aClass3Alarm[5] := 0; END_IF
		
	//IF NewBatch.HoldTank.ActualScaleWeight > NewBatch.HoldTank.FullScaleWeight   						
	//									THEN aClass3Alarm[6] := 1; ELSE aClass3Alarm[6] := 0; END_IF
	
		
// warnings, filter change, refilling of tanks, pre-alarms, etc.

	//IF Ventilation.FILTER_OBSTRUCTED_FAULT	THEN aWarning[0] := 1; ELSE aWarning[0] := 0; END_IF
		
	//IF HMI.Filter2.ChangeOutNeededAlarm = 1		THEN aWarning[1] := 1; ELSE aWarning[1] := 0; END_IF
		
	//IF HMI.Filter3.ChangeOutNeededAlarm = 1		THEN aWarning[2] := 1; ELSE aWarning[2] := 0; END_IF
		
	//IF HMI.Filter4.ChangeOutNeededAlarm = 1		THEN aWarning[3] := 1; ELSE aWarning[3] := 0; END_IF
		
	//IF NewBatch.IngredientsReady = 0			THEN aWarning[4] := 1; ELSE aWarning[4] := 0; END_IF
		
	
// Infos

	IF GVL_Conveyors.ALL_CONVEYORS_IN_CYCLE AND  GVL_CONVEYORS.MOTOR_FAULT_WORD = 0 AND GVL_CONVEYORS.JAM_FAULT_WORD =0 THEN aInfo[0] := 1; ELSE aInfo[0] := 0; END_IF
		
	IF NOT GVL_Conveyors.ALL_CONVEYORS_IN_CYCLE AND  GVL_CONVEYORS.MOTOR_FAULT_WORD = 0 AND GVL_CONVEYORS.JAM_FAULT_WORD =0 THEN aInfo[1] := 1; ELSE aInfo[1] := 0; END_IF
		
	//IF HMI.Filter2.ChangeOutCompleted THEN aInfo[1] := 1; ELSE aInfo[1] := 0; END_IF
END_ACTION

END_PROGRAM

// ---- Machine System/FBs/EventLogger/FB_EventAlarm.TcPOU
FUNCTION_BLOCK FB_EventAlarm
VAR_INPUT 
	bEvent			: BOOL; 
	nEventID		: UDINT; 
	sSource			: STRING; 
END_VAR 
VAR_OUTPUT 
END_VAR
VAR 
	bIsInitalized	: BOOL;
	
	fbSourceInfo 	: FB_TcSourceInfo;
	fbAlarm 		: FB_TCAlarm;
	eventEntry 		: TcEventEntry;
	fbRtEvent 		: R_TRIG;
	fbFtEvent		: F_TRIG;
	
	hr				: HRESULT; 
	hrLastError 	: HRESULT;
	
END_VAR

// Initialization 
	IF NOT bIsInitalized THEN
		bIsInitalized:= TRUE;
		
		eventEntry:= Tc_Events.myAlarmEventClass.x1000; 
		eventEntry.nEventId:= nEventID;
		
		fbSourceInfo.Clear(); 
		fbSourceInfo.sName:= sSource;
		
		hr:= fbAlarm.CreateEx(eventEntry, TRUE, ipSourceInfo:= fbSourceInfo); 
		IF FAILED(hr) THEN
			hrLastError:= hr; 
		END_IF 
	END_IF
	
// event trigger 
	fbRtEvent(CLK:= bEvent); 
	fbFtEvent (CLK:= bEvent);
	
// alarm raised 
	IF  fbRtEvent.Q THEN
		hr:= fbAlarm.Raise(0); 
		IF FAILED(hr) THEN
			hrLastError:= hr; 
		END_IF
	END_IF
	
// alarm cleared 
	IF fbFtEvent.Q THEN
		hr:= fbAlarm.Clear(0, bResetConfirmation:= TRUE); 
		IF FAILED(hr) THEN
			hrLastError:= hr; 
		END_IF 
	END_IF

END_FUNCTION_BLOCK

// ---- Machine System/FBs/EventLogger/FB_EventMessage.TcPOU
FUNCTION_BLOCK FB_EventMessage 
VAR_INPUT 
	bEvent			: BOOL; 
	nEventID		: UDINT; 
	sSource			: STRING; 
END_VAR 
VAR_OUTPUT 
END_VAR 
VAR
	bIsInitalized : BOOL;
	
	fbSourceInfo 	: FB_TcSourceInfo;
	fbMessage 		: FB_TcMessage;
	eventEntry 		: TcEventEntry;
	fbRtEvent		: R_TRIG;
	hr 				: HRESULT;
	hrLastError		: HRESULT;
	
END_VAR

// initialization 
	IF NOT bIsInitalized THEN
		bIsInitalized:= TRUE;
		
		IF nEventID> 16#04FF THEN
			eventEntry:= Tc_Events.myWarningEventClass.x0500; 
		ELSE
			eventEntry:= TC_Events.myInfoEventClass.x0000; 
		END_IF
		
		eventEntry.nEventId:= nEventID;
		fbSourceInfo.Clear(); 
		fbSourceInfo.sName := sSource;
		
		hr:= fbMessage.CreateEx(eventEntry, ipSourceInfo:= fbSourceInfo); 
		IF FAILED (hr) THEN
			hrLastError:= hr; 
		END_IF 
	END_IF
	
// event trigger 
	fbRtEvent (CLK:= bEvent);

// message sent
	IF fbRtEvent.Q THEN
		hr:= fbMessage. Send(0); 
		IF FAILED (hr) THEN
			hrLastError:= hr;
		END_IF 
	END_IF

END_FUNCTION_BLOCK

// ---- Machine System/PRGs/Ventilation.TcPOU
PROGRAM Ventilation
VAR_INPUT
	SettingsArray :  ARRAY[1..2] OF sDatagridVFD;
END_VAR
VAR
	
	VentAreaRequest : BOOL;
	VentAreaTimer 	: TON;
	
	TrenchFanMtr : sVFD;
	FilterBankFanMtr : sVFD;
	
	
	gasSensorNormal  : BOOL;
	gasSensorHigh  : BOOL;
	gasSensorFaulted  : BOOL;
	

	FILTER_CHANGE_NEEDED : BOOL;
	FILTER_OBSTRUCTED_FAULT : BOOL;
	FILTER_OK : BOOL;

	filterCheck : UINT;
	StyreneCheck : UINT;
	ScaledManometer : REAL;
	ScaledStyrene : REAL;
	Results: real;
END_VAR


//setting of the ID strings for the settings page
SettingsArray[1].NameVFD := 'Filter Bank';
SettingsArray[2].NameVFD := 'Trench';

//outputing speed to settings page
SettingsArray[1].CurrentSpeed := FilterBankFanMtr.CurrentSpeed;
SettingsArray[2].CurrentSpeed := TrenchFanMtr.CurrentSpeed;


// Run Vfd Controlled Vent Fans At Optimal Speed Unless Gas Sensor Reads High
IF NOT gasSensorNormal THEN 
	TrenchFanMtr.RunRequest 	:= 1; 
	FilterBankFanMtr.RunRequest := 1; 
    TrenchFanMtr.SpeedRequested 	:= SettingsArray[2].SpeedSetpointLow;
	FilterBankFanMtr.SpeedRequested := SettingsArray[1].SpeedSetpointLow;
	ELSE
	TrenchFanMtr.RunRequest 	:= 1; 
	FilterBankFanMtr.RunRequest := 1; 
    TrenchFanMtr.SpeedRequested 	:= SettingsArray[2].SpeedSetpointHigh;
	FilterBankFanMtr.SpeedRequested := SettingsArray[1].SpeedSetpointHigh;
END_IF


// Manometer for air filters. Analog scaled to 0-100
						
ScaledManometer := ((INT_TO_REAL(GVL_IO.FilterManometer) / 32767 - 0.0)* 100); //* 20; // SCALE OF ANALOG INPUT 0-100

IF ScaledManometer <  49 THEN // ScaledManomter is scaled value from Manometer 0-100. Check that its not to halfway of full range yet.
	filterCheck := 1;
END_IF

IF ScaledManometer >  50 AND ScaledManometer < 80 THEN // ScaledManometer is scaled value from Manometer 0-100. Check if its over halfway of full range yet.
	filterCheck := 2;
END_IF

IF ScaledManometer >  80 OR ScaledManometer < 0 THEN // ScaledManometer is scaled value from Manometer 0-100. Check if its over 80% of full range yet.
	filterCheck := 3;
END_IF
	

CASE filterCheck OF 
     1 : FILTER_OK := TRUE; 
         FILTER_CHANGE_NEEDED := FALSE;
		 FILTER_OBSTRUCTED_FAULT := FALSE; 

     2 : FILTER_CHANGE_NEEDED := TRUE; 
         FILTER_OK := FALSE; 
		 FILTER_OBSTRUCTED_FAULT := FALSE;

	 3 : FILTER_OK := FALSE; 
         FILTER_OBSTRUCTED_FAULT:= TRUE;
		 FILTER_CHANGE_NEEDED := FALSE;
ELSE 
	 FILTER_OK := FALSE;
	 FILTER_OBSTRUCTED_FAULT := FALSE;
	 FILTER_CHANGE_NEEDED := FALSE;
END_CASE;


// Styrene Gas Sensor. Analog scaled to 0-100
//gasSensor := 16000;				
ScaledStyrene := ((INT_TO_REAL(GVL_IO.GasSensor) / 32767 - 0.0)* 100); // SCALE OF ANALOG INPUT 0-100

IF ScaledStyrene <  49 THEN // ScaledStyrene is scaled value from Styrene gas sensor 0-100.  Check that its not to halfway of full range yet.
	StyreneCheck := 1;
END_IF

IF ScaledStyrene >  50 AND ScaledStyrene < 80 THEN // ScaledStyrene is scaled value from Styrene gas sensor 0-100.  Check if its over halfway of full range yet.
	StyreneCheck := 2;
END_IF

IF ScaledStyrene >  80 OR ScaledStyrene < 0 THEN // ScaledStyrene is scaled value from Styrene gas sensor 0-100. Check if its over 80% of full range yet.
	StyreneCheck := 3;
END_IF
	

CASE StyreneCheck OF 
     1 : gasSensorNormal := TRUE; 
         gasSensorHigh := FALSE;
		 gasSensorFaulted := FALSE; 

     2 : gasSensorNormal := FALSE; 
	 	 gasSensorHigh := TRUE;
		 gasSensorFaulted := FALSE;

	 3 : gasSensorNormal := FALSE; 
         gasSensorHigh := FALSE;
		 gasSensorFaulted:= TRUE;
ELSE 
	 gasSensorNormal := FALSE;
	 gasSensorHigh := FALSE;
	 gasSensorFaulted := FALSE;
END_CASE;

// Fault Reset from HMI
	IF  gvl_conveyors.FAULT_RESET	THEN 
		FILTER_OBSTRUCTED_FAULT := FALSE;
		gasSensorFaulted := FALSE;
	END_IF

//timer for a user requested 10 minutes of venting air
//VentAreaRequest := FALSE;
IF VentAreaRequest (*OR gasSensorFaulted OR gasSensorHigh*) THEN // added styrene sensor to conditions to start evacuation of spray area when levels are too high. KT
	VentAreaTimer(IN:=TRUE,PT:=T#10M);
	TrenchFanMtr.RunRequest 	:= 1;
	FilterBankFanMtr.RunRequest := 1;
	TrenchFanMtr.SpeedRequested 	:= SettingsArray[2].SpeedSetpointHigh;
	FilterBankFanMtr.SpeedRequested := SettingsArray[1].SpeedSetpointHigh;
END_IF
IF VentAreaTimer.Q THEN
	VentAreaTimer(IN:=FALSE);
	VentAreaRequest := 0;
END_IF

END_PROGRAM

// ---- Machine System/PRGs/FirstScan.TcPOU
PROGRAM FirstScan
VAR
	SkipFirstScan : BOOL; // You guessed it, this skips the after first scan!
END_VAR

IF SkipFirstScan = FALSE THEN
	
	//Default values for Ventalation
	Ventilation.SettingsArray[2].SpeedSetpointLow 	:= 3000;
	Ventilation.SettingsArray[1].SpeedSetpointLow 	:= 3000;
	Ventilation.SettingsArray[2].SpeedSetpointHigh 	:= 6000;
	Ventilation.SettingsArray[1].SpeedSetpointHigh 	:= 6000;
	
	
	
	SkipFirstScan := TRUE; // keep at bottom
	
END_IF

END_PROGRAM

// ---- CNC/PRG_CNCAxesHandler.TcPOU
PROGRAM PRG_CNCAxesHandler
VAR
	nHliAxisIdx					: INT;				
	fbCNC_Axis					: ARRAY[0..HLI_SYS_AX_MAXIDX] OF FB_CNCAxis;	
	
	nFirstSpindle				: INT := -1;
	fbHandleSpindleTechno		: HLI3_HandleSpindleTechnoGearChange;
	M3,M4,M5,M19				: BOOL;
	MDummy						: BOOL;
	M40, M41, M42, M43, M44, M45: BOOL;
	
	fbAxesError 				: FB_AxesError;
		
	// FB_CNCAxis Sample
	// fbAxis_X 					:  FB_CNCAxis; 
	// stParameter					:  ST_CNC_AX_Parameter;
	// stOptions					:  ST_CNC_AX_Options;
	// stPLCopen					:  ST_CNC_AX_PLCopen;
			
	(*
	fbHandleSpindleTechnoPlcSp	: HLI3_HandleSpindleTechno;
	SM3,SM4,SM5,SM19			: bool; 
	*)
	bCalibrationCam: BOOL;
	fbMoveSpindle: HLI3_MoveSpindle;
END_VAR

(****************************************************************************************)
(* POU:		PRG_AxesHandler                     										*)
(* Type:	PRG																			*)
(* Author: 	TV,MiB                                             							*)
(* Date: 	20.02.2019																	*)
(* Rev.: 	1.6                                               							*)
(* ------------------------------------------------------------------------------------ *)
(* Desc:	Description																	*)
(****************************************************************************************)

fbAxesError(bReset := PLCReset);

(****************************************************************************************)
(*							Release of all reachable axes								*)
(****************************************************************************************)
PLCStatusAxisEnabled := TRUE;   
FOR nHliAxisIdx := 0 TO UDINT_TO_INT(gNrAx-1) DO			
	fbCNC_Axis[nHliAxisIdx](
		nLogAxisNo :=  UINT_TO_INT(gpAx[nHliAxisIdx]^.head.log_ax_nr_r),
		bEnable		:= PLCAxisEnable);
		IF (NOT fbCNC_Axis[nHliAxisIdx].stStatus.bIsEnabled) THEN    // if one axis status is "not enabled" -> reset PLCStatusAxisEnabled
			PLCStatusAxisEnabled := FALSE;
		END_IF
		IF HLI3_CheckAxisValid(nHliAxisIdx) THEN
			IF nFirstSpindle = -1 AND gpAx[nHliAxisIdx]^.ipo_state.spindle_axis_r THEN  (* store HLIIndex of first spindle *)
				nFirstSpindle := nHliAxisIdx;
			END_IF
		END_IF
END_FOR


	// FB_CNCAxis Sample 

	// CNC Axis Options
	
	// stOptions.strPathCompTable;
	// stOptions.bActivateCompTable;
	// stOptions.bProbingSignal;
	// stOptions.bReducedSpeed;
	// stOptions.bReducedSpeedZone1;
	// stOptions.bReducedSpeedZone2;
	// stOptions.bResetCalibration;
	
	// CNC Parameters
			
	// stParameter.bWriteParameter;
	// stParameter.nNumParameters  	:= 2;
	// stParameter.strTempPath		:= 'C:\';
	
	// stParameter.ParamList[0].strName 	:= 'kenngr.swe_pos';
	// stParameter.ParamList[0].strValue 	:= '30000000';

	// stParameter.ParamList[1].strName 	:= 'kenngr.swe_neg';
	// stParameter.ParamList[1].strValue 	:= '0';

	// PLCOpen
	// stPLCopen.nOverride;
	// stPLCopen.bExecuteHoming;
	// stPLCopen.bCamSignal;
	// stPLCopen.bExecuteMoveAbsolute;
	// stPLCopen.bExecuteReset;
	// stPLCopen.fPosition;
	// stPLCopen.fVelocity;
	// stPLCopen.fAcceleration;
	// stPLCopen.fJerk;
	
	(*
	fbAxis_X(
		nLogAxisNo:=1, 
		bEnable:= PLCAxisEnable, 
		bCalibrationCam:= bCalibrationCam, 
		bSetRefOffset:= , 
		fRefOffset:= , 
		bFeedhold:= ,
		stOptions:= stOptions, 
		stParameter:= stParameter, 
		stPLCopen:= stPLCopen, 
		stStatus=> );
*)		
 

(* if there exits spindles use the first one for spindleoverride *)
IF nFirstSpindle <> -1 THEN
	HLI3_SetAxisOverride(nHliAxisIdx:= nFirstSpindle , nOverride:= PLCSpindleOverride *10);

	fbHandleSpindleTechno(
		nHliAxisIdx:=nFirstSpindle , 		
		bIsChannelSpecific:= FALSE, 
		bHandleGearChange := FALSE,		
		nRevolution=> , 
		nPosition=> , 
		bError=> , 
		nErrorId=> , 
		M03:= M3, 
		M04:= M4, 
		M05:= M5, 
		M19:= M19,
		M40 := M40,
		M41 := M41,
		M42 := M42,
		M43 := M43,
		M44 := M44,
		M45 := M45,
		); 
	(* acknowledge all spindle M funnctions immediately *)
	M3 := FALSE;  
	M4 := FALSE;
	M5 := FALSE;
	M19 := FALSE;
	
	
	
	(* Example for starting and stopping a spindle in manual mode in first channel *)
	IF (CNCSystem.Channel[0].ActMode = HLI_IMCM_MANUAL_MODE) THEN 	
		fbMoveSpindle(
			nHliAxisIdx:=nFirstSpindle , 
			nSpeed:= nSpindleRpm ,   (* defined in Global_HMI *)
			bStart:=bSpindleStart, 	 (* defined in Global_HMI *)
			bStop:= bSpindleStop , 	 (* defined in Global_HMI *)
			bBusy=> , 
			bError=> , 
			nErrID=> , 
			sErrText=> );
	END_IF
	IF (bSpindleStart AND NOT fbMoveSpindle.bBusy) THEN 
		bSpindleStart := FALSE;
	END_IF
	IF (bSpindleStop AND NOT fbMoveSpindle.bBusy) THEN 
		bSpindleStop := FALSE;
	END_IF	
	
	
END_IF



(* Howto use plc controlled spindle : *)
(*
fbHandleSpindleTechnoPlcSp(
	nHliAxisIdx:= 0 , 
	nHliChannelIdx:= 0 , 
	bIsChannelSpecific:= TRUE, 
	nLogAxisNoChannelSpecific:= 95 , 
	bHandleGearChange:= FALSE , 
	bChannelReset:= FALSE, 
	nRevolution=> , 
	nPosition=> , 
	bError=> , 
	nErrorId=> , 
	M03:= SM3, 
	M04:= SM4, 
	M05:= SM5, 
	M19:= SM19);
*)

END_PROGRAM

// ---- CNC/PRG_CNCManualMode.TcPOU
PROGRAM PRG_CNCManualMode
VAR
	fbUintUdInt: ARRAY [0..MAX_USED_CHANNEL_IDX] OF FB_Uint_Udint;
	nHandwheel : UINT;		(* increments for handwheel (e.g. EL5101   *)
	nHandWheelBig: UDINT;
	i: INT;
END_VAR


FOR i := 0 TO MAX_USED_CHANNEL_IDX DO
	
	IF (HLI3_CheckChannelValid(i)) THEN

		stManualModeParameter[i].stChannelParameter.nChanIdx						:= i;       (* Channel 1 *)
		stManualModeParameter[i].stChannelParameter.nInc							:= PLCMachineMode[i].ManualMode.nInc * 10;
		stManualModeParameter[i].stChannelParameter.bG200ConfigurationViaPLC		:= TRUE;		
		
		stManualModeParameter[i].stChannelParameter.eManualType						:= UINT_TO_INT(PLCMachineMode[i].ManualMode.nManualTyp);			
		IF (stManualModeParameter[i].stChannelParameter.eManualType = E_CNC_ManualType.Handwheel AND i <> PLCSelectedChannel) THEN	(* if in Handwheel mode and the channel is NOT selected -> leave handwheel mode and change to TippMode*)
			stManualModeParameter[i].stChannelParameter.eManualType						:= E_CNC_ManualType.TippMode;
		END_IF		
		
		stManualModeParameter[i].stChannelParameter.stManualOption.bTrafoActive := PLCMachineMode[i].ManualMode.stManualOption.bTrafoActive;
        stManualModeParameter[i].stChannelParameter.stManualOption.bEcsActive 	:= PLCMachineMode[i].ManualMode.stManualOption.bEcsActive;
        stManualModeParameter[i].stChannelParameter.stManualOption.eZeroOffset 	:= PLCMachineMode[i].ManualMode.stManualOption.eZeroOffset;					
		
		stManualModeParameter[i].stChannelParameter.nHandwheelResolution			:= UDINT_TO_DINT(PLCMachineMode[i].ManualMode.nHwResolution);    (* 0.1 µm /rev (from HMI) *)						
		stManualModeParameter[i].stAxisParameter.stControlUnit[0].nLogAxisNr		:= PLCMachineMode[i].ManualMode.nLogAxisNumber;   (* Log. Achs Nummer *)
		IF stManualModeParameter[i].stAxisParameter.stControlUnit[0].nLogAxisNr = 0 THEN
			stManualModeParameter[i].stAxisParameter.stControlUnit[0].nLogAxisNr := gpCh[i]^.bahn_state.coord_r[0].log_achs_nr_r;
			PLCMachineMode[i].ManualMode.nLogAxisNumber := gpCh[i]^.bahn_state.coord_r[0].log_achs_nr_r;
		END_IF
		stManualModeParameter[i].stAxisParameter.stControlUnit[0].nSpeed			:= LREAL_TO_UDINT(PLCMachineMode[i].ManualMode.nSpeed * 16.666);
		stManualModeControlElements[i].stControlKeys[0].bKeyNeg						:= PLCMachineMode[i].ManualMode.bKeyNeg;
		stManualModeControlElements[i].stControlKeys[0].bKeyPos						:= PLCMachineMode[i].ManualMode.bKeyPos;
		stManualModeControlElements[i].stControlKeys[0].bKeyRapid					:= PLCMachineMode[i].ManualMode.bKeyRapid;
		
		(* the cnc needs an UDINT for handwheel increments, fbUintUdint extends an UInt to an UDINT *)
		(* the resoltion of the handwheel is parameterized in CNC-Task GEO/Manual MDS: (e.g. 400 handwheel inc / handwheel revolution
		
				hr_data[0].hr_aufl_z              400         ( P-MANU-00005 : Handwheel resolution numerator
				hr_data[0].hr_aufl_n                1     	  ( P-MANU-00006 : Handwheel resolution denominator
		*) 
		fbUintUdInt[i](nInSmall := nHandwheel, nBig := nHandWheelBig);
		stManualModeControlElements[i].nHandwheelInc[0] :=  UDINT_TO_DINT(nHandWheelBig);
  END_IF
END_FOR

END_PROGRAM

// ---- CNC/PRG_CNCChannelHandler.TcPOU
PROGRAM PRG_CNCChannelHandler
VAR	
	nChan					: INT;
	nOldSelectedChannel		: UDINT;
	CNCChannel				: ARRAY[0..MAX_USED_CHANNEL_IDX] OF HLI3_CNCChannel;	
	BlockSearch_Channel		: ARRAY[0..MAX_USED_CHANNEL_IDX] OF HLI3_BlockSearch;
	ErrorHandler_Channel	: ARRAY[0..MAX_USED_CHANNEL_IDX] OF FB_ChannelError;
	nChanNo: UDINT;	
	i: INT;	
	stOptions				: ST_CNC_CH_Options;
END_VAR

(****************************************************************************************)
(* POU:		PRG_ChannelHandler                     										*)
(* Type:	PRG																			*)
(* Author: 	HR / TV / MiB                                          						*)
(* Date: 	23.01.11																	*)
(* Last:	29.03.18																	*)
(* Rev.: 	1.6                                              							*)
(* ------------------------------------------------------------------------------------ *)
(* Desc:	Description																	*)
(****************************************************************************************)

(****************************************************************************************)
(*	  Map CNC function selection from HMI to selected channel (and state vice versa)  	*)
(****************************************************************************************)
IF (nOldSelectedChannel <>INT_TO_UDINT(PLCSelectedChannel)) THEN
	PLCChannelSignals.SingleBlock 		:= PLCMachineMode[PLCSelectedChannel].ChannelSignals.SingleBlock;
	PLCChannelSignals.PrgBlockIgnore	:= PLCMachineMode[PLCSelectedChannel].ChannelSignals.PrgBlockIgnore;
	PLCChannelSignals.M01Stop 			:= PLCMachineMode[PLCSelectedChannel].ChannelSignals.M01Stop;
	PLCChannelSignals.Backward 			:= PLCMachineMode[PLCSelectedChannel].ChannelSignals.Backward;
	PLCChannelSignals.FeedHold 			:= PLCMachineMode[PLCSelectedChannel].ChannelSignals.FeedHold;
	nOldSelectedChannel 				:= INT_TO_UDINT(PLCSelectedChannel);
END_IF

PLCMachineMode[PLCSelectedChannel].ChannelSignals.SingleBlock 		:= PLCChannelSignals.SingleBlock;
PLCMachineMode[PLCSelectedChannel].ChannelSignals.PrgBlockIgnore 	:= PLCChannelSignals.PrgBlockIgnore;
PLCMachineMode[PLCSelectedChannel].ChannelSignals.M01Stop 			:= PLCChannelSignals.M01Stop;
PLCMachineMode[PLCSelectedChannel].ChannelSignals.Backward 		:= PLCChannelSignals.Backward;
PLCMachineMode[PLCSelectedChannel].ChannelSignals.FeedHold 		:= PLCChannelSignals.FeedHold;
//PLCMachineMode[PLCSelectedChannel].ChannelSignals.SprayOff 		:= PLCChannelSignals.SprayOff;


stOptions.bReferenceModeStartRequired := FALSE;

FOR i := 0 TO MAX_USED_CHANNEL_IDX DO
		
	nChan := i;	
	IF (HLI3_CheckChannelValid(nChan)) THEN		
		
		(* Error handler for channel  *)
		ErrorHandler_Channel[nChan](nChanIdx			:= nCHan);				
				
		(* Channel interface *)
		CNCChannel[nChan]
			(nChanIdx			:= nChan,							
			 // Operation Mode with VAR_IN_OUT Variables 
			 bModeStandby		:= PLCMachineMode[nChan].Standby,
			 bModeAutomatic		:= PLCMachineMode[nChan].Automatic,
			 bModeManual		:= PLCMachineMode[nChan].Manual,
			 bModeMDI			:= PLCMachineMode[nChan].MDI,	 
			 bModeReference		:= PLCMachineMode[nChan].Homing,
			 // Operation State with VAR_IN_OUT Variables
			 bStateSelect		:= PLCMachineMode[nChan].Select,
			 bStateReady		:= PLCMachineMode[nChan].Ready,
			 bStateStart		:= PLCMachineMode[nChan].Start,
			 bStateStop			:= PLCMachineMode[nChan].Stop,
			 bStateReset		:= PLCMachineMode[nChan].Reset,
			 // Operation Mode with VAR_IN Varaibles, the command is executed with a rising edge 
			 bCmdAutomatic 		:= FALSE,
			 bCmdManual 		:= FALSE,
    		 bCmdReference 		:= FALSE,
    		 bCmdMDI 			:= FALSE,		
			 // Operation State with VAR_IN Varaibles, the command is executed with a rising edge
			 bCmdStart 			:= FALSE,
			 bCmdStop  			:= FALSE,
	         bCmdReset 			:= FALSE,					 			 
			 // EmergencyStop 
			 bEmergencyStop 	:= FALSE,		(* If TRUE the interpolation will be aborted, Signal is no TwinSAFE function !*)
			 // Override 
			 nFeedOverride		:= PLCFeedOverride * 10,
			 nRapidFeedOverride := PLCFeedOverride * 10, 
			 // Special Functions 
			 sProgramName		:= PLCMachineMode[nChan].ProgramName,			 
			 sMDIString			:= PLCMachineMode[nChan].MDIString,
			 bBackwardMotion	:= PLCMachineMode[nChan].ChannelSignals.Backward,
			 bPrgBlockIgnore	:= PLCMachineMode[nChan].ChannelSignals.PrgBlockIgnore,
			 bFeedHold			:= PLCMachineMode[nChan].ChannelSignals.FeedHold,
			 bSingleBlock		:= PLCMachineMode[nChan].ChannelSignals.SingleBlock,
			 bDoSingleBlock		:= PLCMachineMode[nChan].ChannelSignals.DoSingleBlock,
			 bM01Stop			:= PLCMachineMode[nChan].ChannelSignals.M01Stop,
			 nSyntaxCheck		:= PLCMachineMode[nChan].SyntaxCheck.nType,
			 bM30Acknowledgement:= TRUE,
			 
			 // Manual Mode 			 						 
			 stManualModeParameter  	 	 := stManualModeParameter[nChan],
			 stManualModeControlElements	 := stManualModeControlElements[nChan],
			 stManualModeControlElementState := stManualModeControlElementState,
			 // Options
			 stOptions			:= 	stOptions			 			 
			);
			
		
		(* Handle block search *)
		BlockSearch_Channel[nChan]
			(nChanIdx			:= nChan,
			 bStartRead      	:= PLCMachineMode[nChan].BlockSearch.bStartRead,   (* Edge signal *)
			 bStartWrite     	:= PLCMachineMode[nChan].BlockSearch.bStartWrite,  (* Edge signal *)
			 BlockSearch		:= PLCMachineMode[nChan].BlockSearch
			);
		
		CNCSystem.Channel[nChan].ActDistance 	:= DINT_TO_LREAL(BlockSearch_Channel[nChan].coveredDistance_AfterReset) / 10.0;
		CNCSystem.Channel[nChan].ActBlockCount 	:= BlockSearch_Channel[nChan].actualBlockCount_AfterReset;
						
	END_IF
END_FOR

END_PROGRAM

// ---- Machine System/PRGs/CAM_CNC/CNC/myPRG_AxisHomeSwitches_1.TcPOU
PROGRAM myPRG_AxisHomeSwitches_1
VAR
	 
	i: USINT;
	xHomed_X: BOOL;
	xHomed_Y: BOOL;
	xHomed_Z: BOOL;
	xHomed_A: BOOL;
	xHomed_C: BOOL;
	xHi_A: BOOL;
	xLo_A: BOOL;
	xHi_C: BOOL;
	xLo_C: BOOL;
	DriveTorque_A AT %I* : INT;
	Drive_AFree : Bool;
 		
	//fbSetOverride: MC_SetOverride;	
	
	


ncase_A : INT;
ncase_C : INT;


END_VAR


HLI3_SetAxisReferenceCam(nHliAxisIdx := 0, bReferenceCam := bXHomeSwitch);
HLI3_SetAxisReferenceCam(nHliAxisIdx := 1, bReferenceCam := bYHomeSwitch);
HLI3_SetAxisReferenceCam(nHliAxisIdx := 2, bReferenceCam := bZHomeSwitch);
HLI3_SetAxisReferenceCam(nHliAxisIdx := 3, bReferenceCam := DriveTorque_A>700);
HLI3_SetAxisReferenceCam(nHliAxisIdx := 4, bReferenceCam := bCHomeSwitch);


// Below sets all axis positions to zero and sets "homed" flag
//HLI3_SetAxisReferencePosition(bSetRefpos:= bSet, nHliAxisIdx:= 0); // cannot be done in manual mode
//HLI3_SetAxisReferencePosition(bSetRefpos:= bSet, nHliAxisIdx:= 1); // cannot be done in manual mode
//HLI3_SetAxisReferencePosition(bSetRefpos:= bSet, nHliAxisIdx:=2); // cannot be done in manual mode

		
//Axis Home Status i.e. is the axis home
xHomed_X := gpAx[0]^.lr_state.homing_done_r;
xHomed_Y := gpAx[1]^.lr_state.homing_done_r;
xHomed_Z := gpAx[2]^.lr_state.homing_done_r;
xHomed_A := gpAx[3]^.lr_state.homing_done_r;
xHomed_C := gpAx[4]^.lr_state.homing_done_r;

IF xHomed_A = FALSE AND DriveTorque_A>900 THEN ncase_A := 20;
	ELSIF xHomed_A = FALSE AND DriveTorque_A<-600 THEN ncase_A :=30;
		ELSIF xHomed_A = TRUE AND DriveTorque_A > 2000 THEN ncase_A :=20;
			ELSIF xHomed_A =TRUE AND DriveTorque_A<-2000 THEN ncase_A :=30;
	 			ELSE ncase_A :=0;
					//ELSIF Drive_AFree :=FALSE THEN ncase_A :=10;
END_IF


IF xHi_C = FALSE THEN ncase_c := 10;
	ELSIF xLo_C = FALSE THEN ncase_C :=20;
		ELSE ncase_C := 0;
END_IF

IF  DriveTorque_A >700 AND xHomed_A =FALSE AND Global_HMI.PLCMachineMode[0].ManualMode.bKeyNeg = TRUE THEN
	ncase_A :=50;
END_IF
IF DriveTorque_A <-600 AND xHomed_A =FALSE AND Global_HMI.PLCMachineMode[0].ManualMode.bKeyPos = TRUE THEN
	ncase_A :=60;
END_IF
IF  DriveTorque_A >1500 AND xHomed_A =TRUE AND Global_HMI.PLCMachineMode[0].ManualMode.bKeyNeg = TRUE THEN
	ncase_A :=50;
END_IF
IF DriveTorque_A <-1500 AND xHomed_A =TRUE AND Global_HMI.PLCMachineMode[0].ManualMode.bKeyPos = TRUE THEN
	ncase_A :=60;
END_IF
IF xHi_C = FALSE AND Global_HMI.PLCMachineMode[0].ManualMode.bKeyNeg = TRUE THEN
	ncase_C :=30;
END_IF
IF xLo_C = FALSE AND Global_HMI.PLCMachineMode[0].ManualMode.bKeyPos = TRUE THEN
	ncase_C :=40;
END_IF
IF xHi_C AND xLo_C = TRUE THEN 
	ncase_C :=0;
END_IF
CASE ncase_C OF
	0://C Axis Enable
		//gpAx[4]^.ipo_mc_control.override.request_r := 1000;
		gpAx[4]^.ipo_mc_control.override.command_w :=1000;
		gpAx[4]^.ipo_mc_control.override.enable_w := 1;
	10: // C Axis Hi Limit Overtravel
		//gpAx[4]^.ipo_mc_control.override.request_r := 0;
		gpAx[4]^.ipo_mc_control.override.command_w := 0;
		//dialog comment for future to hmi (Hi Limit C Axis)
	20: // C Axis Lo Limit Overtravel
		//gpAx[4]^.ipo_mc_control.override.request_r := 0;
		gpAx[4]^.ipo_mc_control.override.command_w := 0;
		//dialog comment for future to hmi (Lo Limit C Axis)
	30: // C Axis Jog Off Lo Limit
		//gpAx[4]^.ipo_mc_control.override.request_r := 1000;
		gpAx[4]^.ipo_mc_control.override.command_w :=1000;
		gpAx[4]^.ipo_mc_control.override.enable_w := 1;
	40: // C Axis Jog Off Hi Limit
		//gpAx[4]^.ipo_mc_control.override.request_r := 1000;
		gpAx[4]^.ipo_mc_control.override.command_w :=1000;
		gpAx[4]^.ipo_mc_control.override.enable_w := 1;
	90:
END_CASE
CASE ncase_A OF //Limit OverTravel Switches
	0: //A Axis Enable					
		//gpAx[3]^.ipo_mc_control.override.request_r := 1000;
		gpAx[3]^.ipo_mc_control.override.command_w :=1000;
		gpAx[3]^.ipo_mc_control.override.enable_w := 1;
			
	//		IF xHi_A = FALSE THEN ncase:=20;
		//	ELSIF xLo_A = FALSE THEN ncase:=30;
			//	END_IF	
	10: //A axis no movement
		
			           
	20:	//A Axis Hi Limit Switch Overtravel
		//gpAx[3]^.ipo_mc_control.override.request_r := 0;
		gpAx[3]^.ipo_mc_control.override.command_w := 0;		
	30:	//A Axis Lo Limit Switch Overtravel
		//gpAx[3]^.ipo_mc_control.override.request_r := 0;
		gpAx[3]^.ipo_mc_control.override.command_w := 0;		
	
			           
	50:	//enable jog away from Hi limit
		//gpAx[3]^.ipo_mc_control.override.request_r := 1000;
		gpAx[3]^.ipo_mc_control.override.command_w :=1000;
		gpAx[3]^.ipo_mc_control.override.enable_w := 1;	  
	60: //enable jog away from Lo limit
		//gpAx[3]^.ipo_mc_control.override.request_r := 1000;
		gpAx[3]^.ipo_mc_control.override.command_w :=1000;
		gpAx[3]^.ipo_mc_control.override.enable_w := 1;	
		

END_CASE


xHi_A := bHi_A;
xLo_A := bLo_A;
xHi_C := bHi_C;
xLo_C := bLo_C;

END_PROGRAM

// ---- Machine System/PRGs/CAM_CNC/myVE_Vars.TcPOU
PROGRAM myVE_Vars
VAR
//Name each ve_Var lreal as a separate variable if you want to see comments in other sections of program
//NCtoPLC ch[0][pull data from the cnc channel [0]
Spray_X_NctoPLC			:	LREAL;
SPray_Y_NCtoPLC			:	LREAL;
Spray_Z_NCtoPLC			:	LREAL;
SPray_A_NctoPLC			:	LREAL;
Spray_C_NCtoPLC			:	LREAL;
WX1Vert_Dis_NCtoPLC		:	LREAL;
WX1Rot_Dis_NCtoPLC		:	LREAL;
WX1Clamp_Dis_NctoPLc	:	LREAL;
WX2Vert_Dis_NctoPLc		:	LREAL;
WX2Rot_Dis_NCtoPLC		:	LREAL;
WX2Clamp_Dis_NCtoPLC	:	LREAL;
WX3Vert_Dis_NCtoPLC		:	LREAL;
WX3Rot_Dis_NCtoPLC		:	LREAL;
WX3Clamp_Dis_NCtoPLC	:	LREAL;
WX4Vert_Dis_NCtoPLC		:	LREAL;
WX4Rot_Dis_NCtoPLC		:	LREAL;
WX4Clamp_Dis_NctoPLC	:	LREAL;
FlangeHeight_NCtoPLC	: 	LREAL;
SocketHeight_NCtoPLC	: 	LREAL;
TrenchWidth_NCtoPLC		: 	LREAL;
D_NCtoPLC				: 	LREAL;
GratingWidth_NCtoPLC	: 	LREAL;
ribOffset_NCtoPLC		: 	LREAL;
RibLength_NctoPLC		: 	LREAL;
TrenchLength_nctoPLC	: 	LREAL;
GratingLength_NCtoPLC	: 	LREAL;
FirstRib_NCtoPLC		: 	LREAL;
RibSpacing_NCtoPLC		: 	LREAL;
Spare_nctoPLC			: 	LREAL;
SPare2_NCtoPLC			: 	LREAL;


//NCtoPLC ch[1] will need roll channel set as well.  Will prob need each ve used again from ch[0] duplicated for ch[1]

//PLCtoNC
spray_X_PLCtoNC			: LREAL;
Spray_Y_PLCtoNC			: LREAL;
Spray_Z_PLCtoNC			: LREAL;
Spray_A_PLCtoNC			: LREAL;
Spray_C_PLCtoNC			: LREAL;
WX1Vert_PLCtoNC		: LREAL;
WX1Rot_PLCtoNc		: LREAL;
WX1Clamp_PLCtoNC	: LREAL;
WX2Vert_PLCtoNC		: LREAL;
WX2Rot_PLCtoNC		: LREAL;
WX2Clamp_PLCtoNC	: LREAL;
WX3Vert_PLCtoNC		: LREAL;
WX3Rot_PLCtoNC		: LREAL;
WX3Clamp_PLCtoNC	: LREAL;
WX4Vert_PLCtoNC 	: LREAL;
WX4Rot_PLCtoNC		: LREAL;
WX4Clamp_PLCtoNC	: LREAL;

END_VAR

//NCtoPLC [read data from GCode Channel]
	Spray_X_NctoPLc			:= HLI3_GetVEChannelLRealValue(nChanIdx:= 0, nVEIndex:=0, nArrayIndex:=1, bGlobal:=TRUE); //Step_x
	SPray_Y_NCtoPLC			:= HLI3_GetVEChannelLRealValue(nChanIdx:= 0, nVEIndex:=0, nArrayIndex:=2, bGlobal:=TRUE); //Step_Y
	Spray_Z_NCtoPLC			:= HLI3_GetVEChannelLRealValue(nChanIdx:= 0, nVEIndex:=0, nArrayIndex:=3, bGlobal:=TRUE); //Step_z
	SPray_A_NctoPLC			:= HLI3_GetVEChannelLRealValue(nChanIdx:= 0, nVEIndex:=0, nArrayIndex:=4, bGlobal:=TRUE); //Step_a
	Spray_C_NCtoPLC			:= HLI3_GetVEChannelLRealValue(nChanIdx:= 0, nVEIndex:=0, nArrayIndex:=5, bGlobal:=TRUE); //Step_c
	WX1Vert_Dis_NCtoPLC		:= HLI3_GetVEChannelLRealValue(nChanIdx:= 0, nVEIndex:=0, nArrayIndex:=6, bGlobal:=TRUE); //WX1Vert_dis
	WX1Rot_Dis_NCtoPLC 		:= HLI3_GetVEChannelLRealValue(nChanIdx:= 0, nVEIndex:=0, nArrayIndex:=7, bGlobal:=TRUE); //WX1Rot_dis
	WX1Clamp_Dis_NctoPLc	:= HLI3_GetVEChannelLRealValue(nChanIdx:= 0, nVEIndex:=0, nArrayIndex:=8, bGlobal:=TRUE); //WX1Clamp_dis
	WX2Vert_Dis_NctoPLc		:= HLI3_GetVEChannelLRealValue(nChanIdx:= 0, nVEIndex:=0, nArrayIndex:=9, bGlobal:=TRUE); //WX2Vert_dis
	WX2Rot_Dis_NCtoPLC		:= HLI3_GetVEChannelLRealValue(nChanIdx:= 0, nVEIndex:=0, nArrayIndex:=10, bGlobal:=TRUE); //WX2Rot_dis
	WX2Clamp_Dis_NCtoPLC 	:= HLI3_GetVEChannelLRealValue(nChanIdx:= 0, nVEIndex:=0, nArrayIndex:=11, bGlobal:=TRUE); //WX2Clamp_dis
	WX3Vert_Dis_NCtoPLC 	:= HLI3_GetVEChannelLRealValue(nChanIdx:= 0, nVEIndex:=0, nArrayIndex:=12, bGlobal:=TRUE); //WX3Vert_dis
	WX3Rot_Dis_NCtoPLC	 	:= HLI3_GetVEChannelLRealValue(nChanIdx:= 0, nVEIndex:=0, nArrayIndex:=13, bGlobal:=TRUE); //WX3Rot_dis
	WX3Clamp_Dis_NCtoPLC 	:= HLI3_GetVEChannelLRealValue(nChanIdx:= 0, nVEIndex:=0, nArrayIndex:=14, bGlobal:=TRUE); //WX3Clamp_dis
	WX4Vert_Dis_NCtoPLC	 	:= HLI3_GetVEChannelLRealValue(nChanIdx:= 0, nVEIndex:=0, nArrayIndex:=15, bGlobal:=TRUE); //WX4Vert_dis
	WX4Rot_Dis_NCtoPLC	 	:= HLI3_GetVEChannelLRealValue(nChanIdx:= 0, nVEIndex:=0, nArrayIndex:=16, bGlobal:=TRUE); //WX4Rot_dis
	WX4Clamp_Dis_NctoPLC 	:= HLI3_GetVEChannelLRealValue(nChanIdx:= 0, nVEIndex:=0, nArrayIndex:=17, bGlobal:=TRUE); //WX4Clamp_dis
	FlangeHeight_NCtoPLC 	:= HLI3_GetVEChannelLRealValue(nChanIdx:= 0, nVEIndex:=0, nArrayIndex:=18, bGlobal:=TRUE); //FlangeHeight
	SocketHeight_NCtoPLC 	:= HLI3_GetVEChannelLRealValue(nChanIdx:= 0, nVEIndex:=0, nArrayIndex:=19, bGlobal:=TRUE); //SocketHeight
	TrenchWidth_NCtoPLC 	:= HLI3_GetVEChannelLRealValue(nChanIdx:= 0, nVEIndex:=0, nArrayIndex:=20, bGlobal:=TRUE); //TrenchWidth
	D_NCtoPLC			 	:= HLI3_GetVEChannelLRealValue(nChanIdx:= 0, nVEIndex:=0, nArrayIndex:=21, bGlobal:=TRUE); //D
	GratingWidth_NCtoPLC 	:= HLI3_GetVEChannelLRealValue(nChanIdx:= 0, nVEIndex:=0, nArrayIndex:=22, bGlobal:=TRUE); //GratingWidth
	ribOffset_NCtoPLC	 	:= HLI3_GetVEChannelLRealValue(nChanIdx:= 0, nVEIndex:=0, nArrayIndex:=23, bGlobal:=TRUE); //RibOffset
	RibLength_NctoPLC		:= HLI3_GetVEChannelLRealValue(nChanIdx:= 0, nVEIndex:=0, nArrayIndex:=24, bGlobal:=TRUE); //RibLength
	TrenchLength_nctoPLC 	:= HLI3_GetVEChannelLRealValue(nChanIdx:= 0, nVEIndex:=0, nArrayIndex:=25, bGlobal:=TRUE); //TrenchLength
	GratingLength_NCtoPLC 	:= HLI3_GetVEChannelLRealValue(nChanIdx:= 0, nVEIndex:=0, nArrayIndex:=26, bGlobal:=TRUE); //GratingLength
	FirstRib_NCtoPLC	 	:= HLI3_GetVEChannelLRealValue(nChanIdx:= 0, nVEIndex:=0, nArrayIndex:=27, bGlobal:=TRUE); //FirstRib
	RibSpacing_NCtoPLC	 	:= HLI3_GetVEChannelLRealValue(nChanIdx:= 0, nVEIndex:=0, nArrayIndex:=28, bGlobal:=TRUE); //RibSpacing
	Spare_NCtoPLC			:= HLI3_GetVEChannelLRealValue(nChanIdx:= 0, nVEIndex:=0, nArrayIndex:=29, bGlobal:=TRUE); //spare
	Spare2_NCtoPLC		 	:= HLI3_GetVEChannelLRealValue(nChanIdx:= 0, nVEIndex:=0, nArrayIndex:=30, bGlobal:=TRUE); //spare [channel max @100 total]
	
	
//PLCtoNC example [can run these in other pou as necessary - will conflict with GCODE SET Value in channel if used concurrently]
	//HLI3_SetVEChannelLRealValue(nChanIdx:=0,nVEIndex:=0,nArrayIndex:=2, bGlobal:=TRUE, val:=spray_Y_PlctoNC);
	//HLI3_SetVEChannelLRealValue(nChanIdx:=0,nVEIndex:=0,nArrayIndex:=6, bGlobal:=TRUE, val:=WX4Vert_Dis_PLCtoNC);

END_PROGRAM

// ---- Machine System/PRGs/CAM_CNC/myM_CODES.TcPOU
PROGRAM myM_CODES
VAR
	testbit:BOOL;
	rtM2: R_TRIG; 
	rtM30: R_TRIG;
	rtM35: R_TRIG;  //Laser Off
	
	//Spray Gantry MCOdes
		rtM100 : R_TRIG; //spray on  //note current type MOS if delay is too slow for motion use FastMcode or use MNS_SNS type
		rtM101 : R_TRIG; //spray off
		rtM102 : R_TRIG; //Fiber on
		rtM103 : R_TRIG; //Fiber off
		
		rtM910: R_TRIG; //Acetone off
		rtM911: R_Trig; //acetone on
		
	//Roll & Place MCodes
	
	//SD1 & SD2 MCodes
		rtM590 : R_trig; 	//SD1 Move Execute
		rtM591 : R_TRIG; 	//SD2 Move Execute
	//Door MCodes
		rtM600 : R_Trig;	//SD1 Door 	Open
		rtM601 : R_Trig; 	//SD1 Door Close
		rtM602 : R_Trig;	//SD2 Door Open
		rtM603 : R_TRIG;	//SD2 Door Close
		rtM604 : R_TRIG;	//Staging Door Open
		rtM605 : R_TRIG;	//Staging Door Close
		rtM606 : R_TRIG;	//Loading Door Open
		rtM607 : R_TRIG;	//Loading Door Close
		rtM608 : R_TRIG;	//Spray Door Open
		rtM609 : R_TRIG;	//Spray Door Close
		rtM610 : R_TRIG;	//Spray acetone Open
		rtM611 : R_TRIG;	//Spray acetone Close
		rtM612 : R_TRIG;	//Roll acetone Open
		rtM613 : R_TRIG;	//Roll Acetone Close
		rtM614 : R_TRIG;	//Rib Door Open
		rtM615 : R_TRIG;	//Rib Door Close
		rtM616 : R_TRIG;	//Edge Door Open
		rtM617 : R_TRIG; 	//Edge Door Close
		
	//Bogie WX M Codes
		//WX1
		rtM510: R_Trig;	//WX1VertExecute 	[synced A&B]
		rtM511: R_trig; //WX1RotExecute 	[synced A&B]
		rtM512: R_trig; //WX1ClampExecute 	[synced A&B]
		rtM519: R_trig;	//WX1FollowSyncExe	[resync Rot]
		
		//WX2
		rtM520: R_Trig;	//WX2VertExecute 	[synced A&B]
		rtM521: R_trig; //WX2RotExecute 	[synced A&B]
		rtM522: R_trig; //WX2ClampExecute 	[synced A&B]
		rtM529: R_trig;	//WX2FollowSyncExe	[resync Rot]
		
		//WX3
		rtM530: R_Trig;	//WX3VertExecute 	[synced A&B]
		rtM531: R_trig; //WX3RotExecute 	[synced A&B]
		rtM532: R_trig; //WX3ClampExecute	[synced A&B]
		rtM539: R_trig;	//WX3FollowSyncExe	[resync Rot]
		
		//WX4
		rtM540: R_Trig;	//WX4VertExecute 	[synced A&B]
		rtM541: R_trig; //WX4RotExecute 	[synced A&B]
		rtM542: R_trig; //WX4ClampExecute 	[synced A&B]
		rtM549: R_trig;	//WX4FollowSyncExe	[resync Rot]
		
		
	bLaserBeamOn AT %Q* : BOOL;
	bGasOn: BOOL;
	rtReset : R_TRIG;
	iM2Counter : INT;
	iM30Counter : INT;
	iTrunnionMotor : DINT;
END_VAR

(*Use Fast MCode POu and task if these are too slow to respond - Move the code to the other POU and check that it is attached to the Fast MCode Task -  See example*)

rtM35(CLK:= CNCSystem.Channel[0].M[35].bState_rw, Q=> );
IF rtM35.Q THEN 
	bLaserBeamOn := FALSE;
	bSprayOn :=FALSE;
	bGasOn := FALSE;
	CNCSystem.Channel[0].M[35].bState_rw := FALSE;
END_IF

rtM2(CLK:= CNCSystem.Channel[0].M[2].bState_rw, Q=> );
IF rtM2.Q THEN 
	iM2Counter := iM2Counter + 1;
END_IF

rtM30(CLK:= CNCSystem.Channel[0].M[30].bState_rw, Q=> );
IF rtM30.Q THEN 
	iM30Counter := iM30Counter + 1;
END_IF

//add a check in check out variable for each gantry to signal that the SD1 or SD2 rail is in use in a given cell
//Spray Gantry MCodes	
	rtM100(CLK:= CNCSystem.Channel[0].M[100].bState_rw, Q=> ); // spray gun mac valve on
	IF rtM100.Q THEN 
	//	bLaserBeamOn := TRUE;
	//	bGasOn := TRUE;
		GVL_IO.bSprayOn :=TRUE;
		CNCSystem.Channel[0].M[100].bState_rw := FALSE;
	END_IF
	rtM101(CLK:= CNCSystem.Channel[0].M[101].bState_rw, Q=> );	// spray gun mac valve off
	IF rtM101.Q THEN 
	//	bLaserBeamOn := TRUE;
		//bGasOn := TRUE;
		GVL_IO.bSprayOn :=FALSE;
		//test sync req in mdi with this if then using outside of auto rtrig one shot mcode uncomment to use like above and change to MOS type
	(*
		IF TestBit THEN
			CNCSystem.Channel[0].M[101].bState_rw := FALSE;
		END_IF *)
	END_IF
	(*example for flipping Mcode acknowledgment outside of rtrig [useful for aux plc axis or actuators...etc] *)
	IF TestBit THEN
		CNCSystem.Channel[0].M[101].bState_rw := FALSE;
	End_if
	(*end M101 example*)
	
	rtM910 (CLK:=CNCSystem.Channel[0].M[910].bState_rw, Q=>); //M910 aceton mac valve off
	IF rtM910.Q THEN
		GVL_IO.bAceOn := FALSE;
	END_IF
	
	rtM911 (CLK:=CNCSystem.Channel[0].M[911].bState_rw, Q=>);  //M911 acetone mac valve on
	IF rtM911.Q THEN
		GVL_IO.bAceOn := TRUE;
	END_IF
	
//Roll & Place Gantry MCodes

//SD Rails MCodes

//Door MCodes
	(* Add rt and io mapping for each door actuator *)
	
//Bogie MCodes
	rtM510 (Clk:=CNCSystem.Channel[0].M[510].bState_rw, Q=>);
	rtM511 (Clk:=CNCSystem.Channel[0].M[511].bState_rw, Q=>);
	rtM512 (Clk:=CNCSystem.Channel[0].M[512].bState_rw, Q=>);
	rtM519 (Clk:=CNCSystem.Channel[0].M[519].bState_rw, Q=>);
	rtM520 (Clk:=CNCSystem.Channel[0].M[520].bState_rw, Q=>);
	rtM521 (Clk:=CNCSystem.Channel[0].M[521].bState_rw, Q=>);
	rtM522 (Clk:=CNCSystem.Channel[0].M[522].bState_rw, Q=>);
	rtM529 (Clk:=CNCSystem.Channel[0].M[529].bState_rw, Q=>);
	rtM530 (Clk:=CNCSystem.Channel[0].M[530].bState_rw, Q=>);
	rtM531 (Clk:=CNCSystem.Channel[0].M[531].bState_rw, Q=>);
	rtM532 (Clk:=CNCSystem.Channel[0].M[532].bState_rw, Q=>);
	rtM539 (Clk:=CNCSystem.Channel[0].M[539].bState_rw, Q=>);
	rtM540 (Clk:=CNCSystem.Channel[0].M[540].bState_rw, Q=>);
	rtM541 (Clk:=CNCSystem.Channel[0].M[541].bState_rw, Q=>);
	rtM542 (Clk:=CNCSystem.Channel[0].M[542].bState_rw, Q=>);
	rtM549 (Clk:=CNCSystem.Channel[0].M[549].bState_rw, Q=>);
	(* bogie Mcode unlatch and bstate calls are handled in CP_GCode *)
	IF rtm510.Q THEN GVL_M.m510Latch:=1; END_IF
	IF rtm511.Q THEN GVL_M.m511Latch:=1; END_IF
	IF rtm512.Q THEN GVL_M.m512Latch:=1; END_IF
	IF rtm519.Q THEN GVL_M.M519Latch:=1; END_IF
	IF rtm520.Q THEN GVL_M.m520Latch:=1; END_IF
	IF rtm521.Q THEN GVL_M.m521Latch:=1; END_IF
	IF rtm522.Q THEN GVL_M.m522Latch:=1; END_IF
	IF rtm529.Q THEN GVL_M.M529Latch:=1; END_IF
	IF rtm530.Q THEN GVL_M.m530Latch:=1; END_IF
	IF rtm531.Q THEN GVL_M.m531Latch:=1; END_IF
	IF rtm532.Q THEN GVL_M.m532Latch:=1; END_IF
	IF rtm539.Q THEN GVL_M.M539Latch:=1; END_IF
	IF rtm540.Q THEN GVL_M.m540Latch:=1; END_IF
	IF rtm541.Q THEN GVL_M.m541Latch:=1; END_IF
	IF rtm542.Q THEN GVL_M.M542Latch:=1; END_IF
	IF rtm549.Q THEN GVL_M.M549Latch:=1; END_IF

END_PROGRAM

// ---- Machine System/PRGs/mySAFETY.TcPOU
PROGRAM mySAFETY
VAR
	ResetReq	: bool;
	bPlc2TsErrAck AT %Q* : BOOL;
	bPlc2TsRestart AT %Q* : BOOL;
	bPlc2TsSTO AT %Q* : BOOL;
	bInit: BOOL;
	bTsToPlcEstopState AT %I* : BOOL := TRUE;
	bPlc2TsRun AT %Q* : BOOL := TRUE;
	ranint : INT;
	ranbool : BOOL;
	ranbool2 : bool;
END_VAR


bPlc2TsErrAck := FALSE;
IF NOT bInit THEN
	bInit := TRUE;
	bPlc2TsErrAck := TRUE;
END_IF

IF NOT bTsToPlcEstopState THEN
	PLCAxisEnable := FALSE;
END_IF

IF GVL_IO.bEstopPB = FALSE THEN
	GVL_IO.bAceOn := FALSE;
 	GVL_IO.bSprayOn := FALSE;
	GVL_IO.iTrunSig := 0;
END_IF

IF GVL_HMI.ManualMode AND GVL_SAF.DeadmanEnable AND GVL_SAF.EStopOK THEN
	
	GVL_HMI.EnableAll := 1;
	PLCAxisEnable := 1;
	KM1_ContactorOn := 1;
	KM2_ContactorOn := 1;
	
ELSIF GVL_HMI.ManualMode THEN//TEMP REMOVE THIS
	
	GVL_HMI.EnableAll := 1;
	KM1_ContactorOn := 1;
	KM2_ContactorOn := 1;
	
ELSIF GVL_HMI.AutoMode AND GVL_SAF.DeadmanEnable AND GVL_SAF.EStopOK THEN //REMOVE THIS LATER
	
	GVL_HMI.EnableAll := 1;
	PLCAxisEnable := 1;
	KM1_ContactorOn := 1;
	KM2_ContactorOn := 1;
	
ELSE
	
	GVL_HMI.EnableAll := 0;
	PLCAxisEnable := 0;
	KM1_ContactorOn := 0;
	KM2_ContactorOn := 0;

END_IF

(*
IF GVL_HMI.ManualMode AND GVL_SAF.DeadmanEnable AND GVL_SAF.EStopOK THEN
	
	GVL_HMI.EnableAll := 1;
	PLCAxisEnable := 1;
	KM1_ContactorOn := 1;
	KM2_ContactorOn := 1;
	
	ELSE
	
	GVL_HMI.EnableAll := 0;
	PLCAxisEnable := 0;
	KM1_ContactorOn := 0;
	KM2_ContactorOn := 0;

END_IF*)

END_PROGRAM

// ---- Machine System/PRGs/SafetyConnect.TcPOU
PROGRAM SafetyConnect
VAR
END_VAR

IF GVL_HMI.MCR THEN
	IF GVL_Saf.InRun = 0 THEN
		GVL_Saf.Run := 0;
		GVL_Saf.ErrorAcknowledgment :=1;
	ELSE
		GVL_Saf.EStopReset := 1;
	END_IF	
ELSE
	GVL_Saf.EStopReset := 0;
	GVL_Saf.ErrorAcknowledgment :=0;
	GVL_Saf.Run := 1;
END_IF

END_PROGRAM

// ---- Machine System/PRGs/ModeHandle.TcPOU
PROGRAM ModeHandle
VAR
	HoldResinFlag	:	BOOL;	//Flag true after Hold Resin Condition and Until Reset
	HoldMixerFlag	:	BOOL;	//Flag true after Hold Mixer Condition and Until Reset
	StopFlag		:	BOOL;	//Flag true after Stop Condition and Until Reset
	
	testbit: BOOL;
	
END_VAR


(*Mode Handling AUTOMODE = 1 , MANUAL MODE = 2*) 
	IF GVL_HMI.ModeReqAuto =1 AND GVL_HMI.Mode = 0 AND GVL_SAF.EstopOk THEN
		GVL_HMI.Mode :=1;
		GVL_HMI.ModeReqAuto :=0;
	ELSIF GVL_HMI.ModeReqManual = 1 AND GVL_HMI.Mode = 0 AND GVL_SAF.EstopOk THEN
		GVL_HMI.Mode :=2;
		GVL_HMI.ModeReqManual := 0;
	END_IF
	
	IF GVL_HMI.ModeReqNo = 1 OR GVL_SAF.EstopOk = 0  THEN	
		GVL_HMI.Mode := 0;
		GVL_HMI.ModeReqNo := 0;
		testbit := 1;
	END_IF

	IF GVL_HMI.Mode = 0 THEN
		GVL_HMI.NoMode := 1;
		ELSE 
		GVL_HMI.NoMode := 0;
	END_IF
	IF GVL_HMI.Mode = 1 THEN
		GVL_HMI.AutoMode := 1;
		ELSE 
		GVL_HMI.AutoMode := 0;
	END_IF
	IF GVL_HMI.Mode = 2 THEN
		GVL_HMI.ManualMode := 1;
		ELSE 
		GVL_HMI.ManualMode := 0;
	END_IF
(*MCR (Master Control Reset)*)
	//Stop Conditions
	
	IF GVL_HMI.MCR = 1 THEN
	
		WX_CP.WX1(Reset_VI := 1);
		WX_CP.WX2(Reset_VI := 1);
		WX_CP.WX3(Reset_VI := 1);
		WX_CP.WX4(Reset_VI := 1);
	
		GVL_HMI.MCR			:= 0;		
		
	END_IF

END_PROGRAM

// ---- Machine System/PRGs/Bogie/WX_CP.TcPOU
PROGRAM WX_CP
VAR_INPUT
		
	// CPRot 		: ClearpathPosition;
	WX1				: 	BogieComboWX;
	WX2				: 	BogieComboWX;
	WX3				: 	BogieComboWX;
	WX4				: 	BogieComboWX;
END_VAR

VAR
	ResetTrig 	: r_trig;
	Reset_Req 	: BOOL;
	testReset	: BOOL;
	CpTime		: TIME;
	WX4V_Trig 	: r_trig;		//delays the check for target position for a time M540
	WX4R_Trig 	: r_trig; 	//delays the check for target position for a time M541
	WX4C_Trig 	: r_trig;		//delays the check for target position for a time M542
	WX4F_trig 	: r_trig;		//delays the check for target position for a time M549
	WX3V_Trig 	: r_trig;		//delays the check for target position for a time M530
	WX3R_Trig 	: r_trig; 	//delays the check for target position for a time M531
	WX3C_Trig 	: r_trig;		//delays the check for target position for a time M532
	WX3F_trig 	: r_trig;		//delays the check for target position for a time M539
	
		//HMI Visualization Inputs
	VI_Selected_Rail 		: INT;
	VI_Selected_WX 			: INT;
	VI_Selected_Motion 		: STRING;
	VI_Selected_Direction	: INT;
	VI_Stop 				: BOOL;
	VI_Reset 				: BOOL;
	VI_ManualModeReq 		: BOOL;
	VO_Mode 				: BOOL;
	VI_VertJogExecute 		: BOOL;
	VI_SuperJogExecute 		: BOOL;
	VI_JogSlow 				: BOOL;
	VI_CW 					: BOOL;
	
	//HMI Visualization Inputs
	VO_Selected_Rail 		: INT;
	VO_Selected_WX 			: INT;
	VO_Selected_Motion 		: INT;
	VO_Selected_Direction	: INT;


	MDICase_0 		: INT;	//Spray Channel Gcode
	MDICase_1 		: INT; 	//Roll Channel GCode
	ClampHomeCase	: INT;

	//CPVert1	: 	ClearpathPositionLinPPR ;
	BogStart	: BOOL;
	EnableM		: BOOL;	//motor enable

	Stop 		: BOOL;
	BeginHoming : BOOL;
	degReq		: REAL;

	enableTest 	 AT %Q*	: BOOL;
	BoutTest	 AT %Q* : BOOL;
	AoutTest	 AT %Q* : BOOL;
	CPvert2Hi_NO AT %I* : BOOL;
	CPvert2Lo_NO AT %I* : BOOL;

END_VAR
VAR PERSISTENT
	cprot1Hi		: INT;			//software limit high
	cprot1Lo		: INT;			//software limit low
	CPVert1Lo		: INT := -125;	//software limit Low
	CPVert1Hi		: INT := 0;		//software limit high
	CPVert2Lo		: INT := -125;	//software limit Low
	CPVert2Hi		: INT := 0;		//software limit high
	Vert_ATrack5	: REAL;			//track the distance when not homed
	Vert_BTrack5	: REAL;			//track the distance when not homed
END_VAR

ResetTrig(Clk:=WX4.Reset_VI, Q=>);
CpTime:=T#100MS;
WX3V_Trig(clk:=WX3.VertInTargetPos_PO);
WX3R_Trig(clk:=WX3.RotInTargetPos_PO);
WX3C_Trig(clk:=WX3.ClampInTargetPos_PO);
WX3F_Trig(clk:=WX3.RotInTargetPos_PO);

IF ResetTrig.Q THEN TestReset:=1; END_IF

//WX1(Mode_PI:= GVL_HMI.Mode, (*Reset_VI:=TestReset,*)VertVE:=myVE_Vars.WX1Vert_Dis_NCtoPLC,RotVE:=myVE_Vars.WX1Rot_Dis_NCtoPLC,ClampVE:=myVE_Vars.WX1Clamp_Dis_NCtoPLC, Vert_A_CI:=GVL_CP.WX1A_CP1_CIn ,Vert_B_CI:=GVL_CP.WX1B_CP1_CIn ,Clamp_A_CI:= GVL_CP.WX1A_CP3_CI,Clamp_B_CI:= GVL_CP.WX1B_CP3_CI ,Rot_A_CI:=GVL_CP.WX1A_CP2_CIn, Rot_B_CI:=GVL_CP.WX1B_CP2_CI, PowerOn_PI:=GVL_HMI.EnableAll,Stop_pi:=stop ,VertSyncTolerance_CI :=20, RotSyncTolerance_CI:=10);

WX2(Mode_PI:= GVL_HMI.Mode, Reset_VI:=GVL_HMI.MCR, VertVE:=myVE_Vars.WX2Vert_Dis_NCtoPLC,RotVE:=myVE_Vars.WX2Rot_Dis_NCtoPLC,ClampVE:=myVE_Vars.WX2Clamp_Dis_NCtoPLC, Vert_A_CI:=GVL_CP.WX2A_CP1_CI ,Vert_B_CI:=GVL_CP.WX2B_CP1_CIn ,Clamp_A_CI:= GVL_CP.WX2A_CP3_CI,Clamp_B_CI:= GVL_CP.WX2B_CP3_CI ,Rot_A_CI:=GVL_CP.WX2A_CP2_CI, Rot_B_CI:=GVL_CP.WX2B_CP2_CI, PowerOn_PI:=GVL_HMI.EnableAll,Stop_pi:=stop ,VertSyncTolerance_CI :=20, RotSyncTolerANce_CI:=10);
WX3(Mode_PI:= GVL_HMI.Mode, (*Reset_VI:=TestReset,*)VertVE:=myVE_Vars.WX3Vert_Dis_NCtoPLC,RotVE:=myVE_Vars.WX3Rot_Dis_NCtoPLC,ClampVE:=myVE_Vars.WX3Clamp_Dis_NCtoPLC, Vert_A_CI:=GVL_CP.WX3A_CP1_CI ,Vert_B_CI:=GVL_CP.WX3B_CP1_CI ,Clamp_A_CI:= GVL_CP.WX3A_CP3_CI,Clamp_B_CI:= GVL_CP.WX3B_CP3_CI ,Rot_A_CI:=GVL_CP.WX3A_CP2_CI, Rot_B_CI:=GVL_CP.WX3B_CP2_CI, PowerOn_PI:=GVL_HMI.EnableAll,Stop_pi:=stop ,VertSyncTolerance_CI :=20, RotSyncTolerance_CI:=10);
WX4(Mode_PI:= GVL_HMI.Mode, (*Reset_VI:=TestReset,*)VertVE:=myVE_Vars.WX4Vert_Dis_NCtoPLC,RotVE:=myVE_Vars.WX4Rot_Dis_NCtoPLC,ClampVE:=myVE_Vars.WX4Clamp_Dis_NCtoPLC, Vert_A_CI:=GVL_CP.WX4A_CP1_CI ,Vert_B_CI:=GVL_CP.WX4B_CP1_CI ,Clamp_A_CI:= GVL_CP.WX4A_CP3_CI,Clamp_B_CI:= GVL_CP.WX4B_CP3_CI ,Rot_A_CI:=GVL_CP.WX4A_CP2_CI, Rot_B_CI:=GVL_CP.WX4B_CP2_CI, PowerOn_PI:=GVL_HMI.EnableAll,Stop_pi:=stop ,VertSyncTolerance_CI :=20, RotSyncTolerANce_CI:=10);
//handle visualiation selection to not have multiple axis selected
	IF VI_Selected_WX <> 1 THEN WX1.AxisSel_VI:=0; END_IF
	IF VI_Selected_WX <> 2 THEN WX2.AxisSel_VI:=0; END_IF
	IF VI_Selected_WX <> 3 THEN WX3.AxisSel_VI:=0; END_IF
	IF VI_Selected_WX <> 4 THEN WX4.AxisSel_VI:=0; END_IF
//cprot(In:=GVL_CP.WX4A_CP2_CI,Poweron_PI:=EnableM,Stop_PI:=stop,);

//WX AutoMode
IF GVL_HMI.Mode = 1 AND PRG_CNCChannelHandler.CNCChannel[0].pChannel^.ActMode = 3  THEN  //change bogstart to a channel based variable for mdi
	//cancel move or pause move [may want to capture current aux move in future to continue on after hitting start]
	IF PRG_CNCChannelHandler.CNCChannel[0].pChannel^.ActStateString ='Hold' THEN
		MDICase_0:=90; //go to stop condition for aux axes in chan[0] during cnc hmi stop command
	END_IF
	CASE MDICase_0 OF (* channel[0] spray *)
	0: //read in VE Variable Requests from MDI Channel
		IF GVL_HMI.Mode =1 AND PRG_CNCChannelHandler.CNCChannel[0].currentmode = 3 THEN //may add a check bit to look for channel selection [cnc auto, mdi, manual] and to confirm for ch 0
			//add in all the other WX
			 //read in variable from Gcode
				
			
			MDICase_0:=10;
		END_IF
	10://Move MDI on MCode Click [can be multiple types depending on if line was called togther on Gcode]
		//WX1
			IF WX1.VertReadyForMove_PO AND WX1.VertInTargetPos_PO AND GVL_M.M510Latch THEN //if in MDI MODE for CP and on M510 use
				WX1.VertDisReq_PI 	:= LREAL_TO_INT(myVE_Vars.WX1Vert_Dis_NCtoPLC);
				WX1.bMoveVert_PI :=1;
				GVL_M.M510Latch:=0;
			END_IF
			(* resync the rot follower if needed via gcode mdi *)
			IF GVL_M.M519Latch  THEN
				WX1.bFollowerIdleDisengage :=1;
				WX1.JogSeparate_VI :=1;
				WX1.Reset_VI:=1;
				WX1.RotDegReq_PI := LREAL_TO_INT(WX1.Rot_A.Out.DistancePos_PO);
				WX1.bMoveRot_PI:=1;
				GVL_M.M519Latch:=0;
			END_IF
			IF WX1.RotReadyForMove_PO AND WX1.RotInTargetPos_PO AND GVL_M.M511Latch THEN
				WX1.RotDegReq_PI 	:= LREAL_TO_INT(myVe_Vars.WX1Rot_Dis_NCtoPLC);
				WX1.bMoveRot_PI := 1;
				GVL_M.M511Latch:=0; 
			END_IF
			IF WX1.ClampReadyForMove_PO AND WX1.ClampinTargetPos_PO AND GVL_M.M512Latch THEN
				WX1.ClampDisReq_PI	:= LREAL_TO_INT(myVe_Vars.WX1Clamp_Dis_NctoPLC);
				WX1.bMoveClamp_PI :=1;
				GVL_M.M512Latch:=0;
			END_IF
		//WX2
			IF Wx2.VertReadyForMove_PO AND Wx2.VertInTargetPos_PO AND GVL_M.M520Latch THEN //if in MDI MODE for CP and on M510 use
				Wx2.VertDisReq_PI 	:= LREAL_TO_INT(myVE_Vars.Wx2Vert_Dis_NCtoPLC);
				WX2.bMoveVert_PI :=1;
				GVL_M.M520Latch:=0;
			END_IF
			(* resync the rot follower if needed via gcode mdi *)
			IF GVL_M.M529Latch  THEN
				WX2.bFollowerIdleDisengage :=1;
				WX2.JogSeparate_VI :=1;
				WX2.Reset_VI:=1;
				WX2.RotDegReq_PI := LREAL_TO_INT(WX2.Rot_A.Out.DistancePos_PO);
				WX2.bMoveRot_PI:=1;
				GVL_M.M529Latch:=0;
			END_IF
			IF Wx2.RotReadyForMove_PO AND Wx2.RotInTargetPos_PO AND GVL_M.M521Latch THEN
				WX2.RotDegReq_PI 	:= LREAL_TO_INT(myVe_Vars.WX2Rot_Dis_NCtoPLC);
				WX2.bMoveRot_PI := 1;
				GVL_M.M521Latch:=0; 
			END_IF
			IF WX2.ClampReadyForMove_PO AND WX2.ClampinTargetPos_PO AND GVL_M.M522Latch THEN
				WX2.ClampDisReq_PI	:= LREAL_TO_INT(myVe_Vars.WX2Clamp_Dis_NctoPLC);
				Wx2.bMoveClamp_PI :=1;
				GVL_M.M522Latch:=0;
			END_IF
		//WX3
			IF WX3.VertReadyForMove_PO AND WX3.VertInTargetPos_PO AND GVL_M.M530Latch  THEN //if in MDI MODE for CP and on M510 use
				WX3.VertDisReq_PI 	:= LREAL_TO_INT(myVE_Vars.WX3Vert_Dis_NCtoPLC);
				WX3.bMoveVert_PI :=1;
				GVL_M.M530Latch:=0;
			END_IF
			(* resync the rot follower if needed via gcode mdi *)
			IF GVL_M.M539Latch  THEN
				WX3.bFollowerIdleDisengage :=1;
				WX3.JogSeparate_VI :=1;
				WX3.Reset_VI:=1;
				WX3.RotDegReq_PI := LREAL_TO_INT(WX3.Rot_A.Out.DistancePos_PO);
				WX3.bMoveRot_PI:=1;
				GVL_M.M539Latch:=0;
			END_IF
			IF WX3.RotReadyForMove_PO AND WX3.RotInTargetPos_PO AND GVL_M.M531Latch  THEN
				WX3.RotDegReq_PI 	:= LREAL_TO_INT(myVe_Vars.WX3Rot_Dis_NCtoPLC);
				WX3.bMoveRot_PI := 1;
				GVL_M.M531Latch:=0; 
			END_IF
			IF WX3.ClampReadyForMove_PO AND WX3.ClampinTargetPos_PO AND GVL_M.M532Latch THEN
				WX3.ClampDisReq_PI	:= LREAL_TO_INT(myVe_Vars.WX3Clamp_Dis_NctoPLC);
				WX3.bMoveClamp_PI :=1;
				GVL_M.M532Latch:=0;
			END_IF
		//WX4
			IF WX4.VertReadyForMove_PO AND WX4.VertInTargetPos_PO AND GVL_M.M540Latch  THEN //if in MDI MODE for CP and on M510 use
				WX4.VertDisReq_PI 	:= LREAL_TO_INT(myVE_Vars.WX4Vert_Dis_NCtoPLC);
				WX4.bMoveVert_PI :=1;
				GVL_M.M540Latch:=0;
			END_IF
			(* resync the rot follower if needed via gcode mdi *)
			IF GVL_M.M549Latch  THEN
				WX4.bFollowerIdleDisengage :=1;
				WX4.JogSeparate_VI :=1;
				WX4.Reset_VI:=1;
				WX4.RotDegReq_PI := LREAL_TO_INT(WX4.Rot_A.Out.DistancePos_PO);
				WX4.bMoveRot_PI:=1;
				GVL_M.M549Latch:=0;
			END_IF
			IF WX4.RotReadyForMove_PO AND WX4.RotInTargetPos_PO AND GVL_M.M541Latch THEN
				WX4.RotDegReq_PI 	:= LREAL_TO_INT(myVe_Vars.WX4Rot_Dis_NCtoPLC);
				WX4.bMoveRot_PI := 1;
				GVL_M.M541Latch:=0; 
			END_IF
			IF WX4.ClampReadyForMove_PO AND WX4.ClampinTargetPos_PO AND GVL_M.M542Latch THEN
				WX4.ClampDisReq_PI	:= LREAL_TO_INT(myVe_Vars.WX4Clamp_Dis_NctoPLC);
				WX4.bMoveClamp_PI :=1;
				GVL_M.M542Latch:=0;
			END_IF
		//add timer buffer if needed
		MDICase_0:=11; //go to wait for plc ack
	11: MDICase_0:=12;
	12: MDICase_0:=15;
	15: //Wait for Move to complete before acknowledgme
	//WX1
		IF WX1.VertReadyForMove_PO AND WX1.VertInTargetPos_PO THEN
			CNCSystem.Channel[0].M[510].bState_rw := FALSE; //M510 Ack to CNC - if it was triggered after reaching position
		END_IF
		IF WX1.RotReadyForMove_PO AND WX1.RotInTargetPos_PO THEN
			CNCSystem.Channel[0].M[511].bState_rw := FALSE; //M511 Ack to CNC
		END_IF
		IF WX1.ClampReadyForMove_PO AND WX1.ClampInTargetPos_PO THEN
			CNCSystem.Channel[0].M[512].bState_rw := FALSE; //M512 Ack to CNC
		END_IF
		IF ABS (WX1.Rot_A.Out.DistancePos_PO-WX1.Rot_B.Out.DistancePos_PO) <= WX1.RotSyncTolerance_CI THEN 
			CNCSystem.Channel[0].M[519].bState_rw := FALSE; //M519 Ack to CNC
			WX1.bFollowerIdleDisengage :=0;
			WX1.JogSeparate_VI :=0;
			WX1.Reset_VI:=0;
		END_IF
		
	//WX2
		IF WX2.VertReadyForMove_PO AND WX2.VertInTargetPos_PO THEN
			CNCSystem.Channel[0].M[520].bState_rw := FALSE; //M520 Ack to CNC - if it was triggered after reaching position
		END_IF
		IF WX2.RotReadyForMove_PO AND WX2.RotInTargetPos_PO THEN
			CNCSystem.Channel[0].M[521].bState_rw := FALSE; //M521 Ack to CNC
		END_IF
		IF WX2.ClampReadyForMove_PO AND WX2.ClampInTargetPos_PO THEN
			CNCSystem.Channel[0].M[522].bState_rw := FALSE; //M522 Ack to CNC
		END_IF
		IF ABS (WX2.Rot_A.Out.DistancePos_PO-WX2.Rot_B.Out.DistancePos_PO) <= WX2.RotSyncTolerance_CI THEN 
			CNCSystem.Channel[0].M[529].bState_rw := FALSE; //M529 Ack to CNC
			WX2.bFollowerIdleDisengage :=0;
			WX2.JogSeparate_VI :=0;
			WX2.Reset_VI:=0;
		END_IF
		
	//WX3
		IF WX3.VertReadyForMove_PO AND WX3.VertIn_M_Pos_PO THEN
			CNCSystem.Channel[0].M[530].bState_rw := FALSE; //M530 Ack to CNC - if it was triggered after reaching position
		END_IF
		IF WX3.RotReadyForMove_PO AND WX3.RotIn_M_Pos_PO THEN
			CNCSystem.Channel[0].M[531].bState_rw := FALSE; //M531 Ack to CNC
		END_IF
		IF WX3.ClampReadyForMove_PO AND WX3.ClampIn_M_Pos_PO THEN
			CNCSystem.Channel[0].M[532].bState_rw := FALSE; //M532 Ack to CNC
		END_IF
		IF ABS (WX3.Rot_A.Out.DistancePos_PO-WX3.Rot_B.Out.DistancePos_PO) <= WX3.RotSyncTolerance_CI THEN 
			CNCSystem.Channel[0].M[539].bState_rw := FALSE; //M539 Ack to CNC
			WX3.bFollowerIdleDisengage :=0;
			WX3.JogSeparate_VI :=0;
			WX3.Reset_VI:=0;
		END_IF
		
	//WX4
		IF WX4.VertReadyForMove_PO AND WX4.VertIn_M_Pos_PO THEN
			CNCSystem.Channel[0].M[540].bState_rw := FALSE; //M540 Ack to CNC - if it was triggered after reaching position
		END_IF
		IF WX4.RotReadyForMove_PO AND WX4.RotIn_M_Pos_PO THEN
			CNCSystem.Channel[0].M[541].bState_rw := FALSE; //M541 Ack to CNC
		END_IF
		IF WX4.ClampReadyForMove_PO AND WX4.ClampIn_M_Pos_PO THEN
			CNCSystem.Channel[0].M[542].bState_rw := FALSE; //M542 Ack to CNC
		END_IF
		IF ABS (WX4.Rot_A.Out.DistancePos_PO-WX4.Rot_B.Out.DistancePos_PO) <= WX4.RotSyncTolerance_CI THEN 
			CNCSystem.Channel[0].M[549].bState_rw := FALSE; //M549 Ack to CNC
			WX4.bFollowerIdleDisengage :=0;
			WX4.JogSeparate_VI :=0;
			WX4.Reset_VI:=0;
		END_IF
		MDICase_0:=20;
	20: MDICase_0 :=0;
	90: //stop condition for cnc stop button
		stop:=1;
		MDICase_0:=91;
	91: //await reset or start cmd from cnc/main hmi
		
		IF PRG_CNCChannelHandler.CNCChannel[0].pChannel^.ActStateString ='Active' OR GVL_HMI.MCR THEN
			MDICase_0:=0;
			Stop:=0;
		END_IF
		
	END_CASE
END_IF

END_PROGRAM

// ---- Machine System/PRGs/Bogie/BogieComboWX.TcPOU
FUNCTION_BLOCK BogieComboWX
VAR_INPUT
	//Configuration Inputs
	VertSyncTolerance_CI 	: INT;
	RotSyncTolerance_CI		: INT;
	Vert_A_CI				: CpABS_CI;
	Vert_B_CI				: CpABS_CI;
	Clamp_A_CI				: CpABS_CI;
	Clamp_B_CI				: CpABS_CI;
	Rot_A_CI				: CpABS_CI;
	Rot_B_CI				: CpABS_CI;
	//VI (visualization input/hmi input)
	AxisSel_VI				: INT;		//selection of Axis for jog[0=none, 1=Vert_Sync, 2=Rot_Sync, 3=Clamp_Sync, 4=Vert_A, 5=Vert_B, 6=Rot_A, 7=Rot_B, 8=Clamp_A, 9=Clamp_B]
	Reset_VI				: BOOL;		//reset button	
	ReSync_VI				: BOOL;		//request resync of dual axis	
	JogSeparate_VI			: BOOL;		//Jog Separate
	A_Select_VI				: BOOL;		//A selected
	B_Select_VI				: BOOL;		//B selectd
	JogNeg_VI				: BOOL;
	JogPos_VI				: BOOL;
	SJogNeg_VI				: BOOL;
	SJogPos_VI				: BOOL;
	JogVertAExecute_VI		: BOOL;		//Call manual vert move method if true
	JogVertBExecute_VI		: BOOL;		//Call manual vert move method if true
	JogClampAExecute_VI		: BOOL;		//Call manual Clamp move method if true
	JogClampBExecute_VI		: BOOL;		//Call manual Clamp move method if true
	JogRotAExecute_VI		: BOOL;		//Call manual Rot Move method if true
	JogRotBExecute_VI		: BOOL;		//Call manual Rot Move method if true
	SyncVertSuperJogExecute_VI	: BOOL;		//sync superjog vert manual move action bit
	SyncRotSuperJogExecute_VI	: BOOL;
	SyncClampSuperJogExecute_VI	: BOOL;
	SuperJogMode_VI			: BOOL;		//Superjog mode enable bit
	(* just use the vert_A. etc
	VertASuperJog_VI		: BOOL;
	VertBSuperJog_VI		: BOOL;	
	RotASuperJog_VI			: BOOL;
	RotBSuperJog_VI			: BOOL;
	ClampASuperJog_VI		: BOOL;
	ClampBSuperJog_VI		: BOOL;	
	*)
	JogSlow_VI				: BOOL;		//slow manual move [default to 1 on init]
	CW_VI					: BOOL;		//Set Direction for requested move (does not apply to absolute move) True = Clockwise
	SyncVertJogExecute_VI 	: BOOL;
	SyncClampJogExecute_VI 	: BOOL;
	SyncRotJogExecute_VI	: BOOL;

	//Program Inputs
	Mode_PI					: INT;		//1:auto, 0:no mode, 2:manual
	ReSync_PI				: BOOL; 	//trigger this to begin a resync process [used after slippage or after individual jogging]
	PowerOn_PI				: BOOL;
	VertDisReq_PI			: INT;
	bMoveVert_PI			: BOOL;		//trigger command for ABSMove [vert]
	bMoveVert_A_PI			: BOOL;	
	bMoveVert_B_PI			: BOOL;
	ClampDisReq_PI			: INT;
	bMoveClamp_PI			: BOOL;		//trigger command for ABSMove [clamp]
	RotDegReq_PI			: INT;
	bMoveRot_PI				: BOOL;		//Trigger command for ABSMove [rot]
	bFollowerIdleDisengage	: BOOL;		//Disconnect sync when idler motor not engaged
	HomeWithPartStart_PI	: BOOL;		//set this true in program with oneshot to start homing, do not hold true in program as FB.Home() will continue to start at step 1
	SyncAbsDisReq_PI		: REAL;
	Stop_PI					: BOOL;		//stop command from program
	bPresetMoveTrigger		: BOOL;		//JOSEPHBARTONCHANGE3-28-2023 This allows for tracking when it is a preset position move
		//VE Req Vars
		ClampVE	: LREAL;
		RotVE	: LREAL;
		VertVE	: LREAL;
	//Field Inputs
	PartPres_A_Hi			: BOOL;
	PartPres_A_Lo			: BOOL;
	PartPres_B_Hi			: BOOL;
	PartPres_B_Lo			: BOOL;
	
	Vert_A					: ClearpathPositionABS;
	Vert_B					: ClearpathPositionABS;
	Clamp_A 				: ClearpathPositionABS;
	Clamp_B					: ClearpathPositionABS;
	Rot_A					: ClearpathPositionABS;		//may need to change to a degree based system
	Rot_B					: ClearpathPositionABS;		//may need to change to a degree based system
	
END_VAR
VAR_OUTPUT
	//Program OutPuts
	Homed_PO				: BOOL;	
	VertReadyForMove_PO		: BOOL;		//ready for vert ABSMove Command
	VertInPosition_PO		: BOOL;		//both vert a and b are in req position
	VertInTargetPos_PO		: BOOL;		//current pos is at last req pos
	VertIn_M_Pos_PO			: BOOL;		//out.pos matches req VE Pos
	VertMoving_PO			: BOOL;		//vert moving in auto mode
	MCodeRec_Vert			: BOOL;		//MCode Command Received [vert]
	McodeComp_vert			: BOOL;		//MCode Command complete [vert]

	RotReadyForMove_PO		: BOOL;		//ready for rot ABSMove command
	RotInPosition_PO		: BOOL;
	RotInTargetPos_PO		: BOOL;
	RotIn_M_Pos_PO			: BOOL; 	//out.pos matches req VE Pos
	RotMoving_PO			: BOOL;		//rot moving in auto mode
	MCodeRec_Rot			: BOOL;		//MCode Command Received [rot]
	MCodeComp_Rot			: BOOL;		//Mcode Command Complet [rot]
	
	ClampReadyForMove_PO	: BOOL;		//ready for clamp absmove command
	ClampInPosition_PO		: BOOL;
	ClampInTargetPos_PO		: BOOL;
	ClampIn_M_Pos_PO		: BOOL;		//out.pos matches req VE Pos
	ClampMoving_PO			: BOOL;		//clamp moving in auto mode
	MCodeRec_Clamp			: BOOL;		//MCode Command Received [clamp]
	MCodeComp_Clamp			: BOOL;		//MCode Command Completed [clamp]
	Msg						: STRING;	//debug message
	Msg_Mode				: STRING; 	//mode message (what mode)
	//Visualization Outputs
	ErrorMsg_VO				: STRING;
	SyncVertMsg_VO			: STRING;
	SyncRotMsg_VO			: STRING;
	SyncClampMsg_VO			: STRING;
	ReadyForMoveMSg_VO		: STRING;
	
END_VAR
VAR
	synctestbit				: BOOL;
    SyncVertCase			: INT;
	SyncRotCase				: INT;
	SyncClampCase			: INT;
END_VAR

//initialize the fb for bogie clearpaths bog[1-4 (vert, rot, clamp)
Clamp_A	(IN:=Clamp_A_CI, Mode_PI:=Mode_PI,VEReq:=ClampVE, DisReq_VI:=ClampDisReq_PI, Poweron_PI:=Poweron_pi, Stop_PI:=Stop_PI, Reset_VI:=Reset_VI, SuperJogMode_VI:=SuperJogMode_VI, JogExecute_VI:=JogClampAExecute_VI, JogSlow_VI:=JogSlow_VI, CW_VI:=CW_VI);
Clamp_B	(IN:=Clamp_B_CI, Mode_PI:=Mode_PI,VEReq:=ClampVE, DisReq_VI:=ClampDisReq_PI, Poweron_PI:=Poweron_pi, Stop_PI:=Stop_PI, Reset_VI:=Reset_VI, SuperJogMode_VI:=SuperJogMode_VI, JogExecute_VI:=JogClampBExecute_VI, JogSlow_VI:=JogSlow_VI, CW_VI:=CW_VI);
Vert_A	(IN:=Vert_A_CI,  Mode_PI:=Mode_PI,VEReq:=VertVE,  DisReq_VI:=VertDisReq_PI,  Poweron_PI:=Poweron_pi, Stop_PI:=Stop_PI, Reset_VI:=Reset_VI, SuperJogMode_VI:=SuperJogMode_VI, JogExecute_VI:=JogVertAExecute_VI,  JogSlow_VI:=JogSlow_VI, CW_VI:=CW_VI);
Vert_B	(IN:=Vert_B_CI,  Mode_PI:=Mode_PI,VEReq:=VertVE,  DisReq_VI:=VertDisReq_PI,  Poweron_PI:=Poweron_pi, Stop_PI:=Stop_PI, Reset_VI:=Reset_VI, SuperJogMode_VI:=SuperJogMode_VI, JogExecute_VI:=JogVertBExecute_VI,  JogSlow_VI:=JogSlow_VI, CW_VI:=CW_VI);
Rot_A	(IN:=Rot_A_CI, 	 Mode_PI:=Mode_PI,VEReq:=RotVE,   DisReq_VI:=RotDegReq_PI,   Poweron_PI:=Poweron_PI, Stop_PI:=Stop_PI, Reset_VI:=Reset_VI, SuperJogMode_VI:=SuperJogMode_VI, JogExecute_VI:=JogRotAExecute_VI,   JogSlow_VI:=JogSlow_VI, CW_VI:=CW_VI);
Rot_B	(IN:=Rot_B_CI, 	 Mode_PI:=Mode_PI,VEReq:=RotVE,   DisReq_VI:=RotDegReq_PI,   Poweron_PI:=Poweron_PI, Stop_PI:=Stop_PI, Reset_VI:=Reset_VI, SuperJogMode_VI:=SuperJogMode_VI, JogExecute_VI:=JogRotBExecute_VI,   JogSlow_VI:=JogSlow_VI, CW_VI:=CW_VI);
//intialize the fb for bogie servo axis 1 and axis 2 in main pou	
//enable motors with enable hmi variable
IF Vert_A.Out.Homed_PO=0 OR Vert_B.Out.Homed_PO=0 OR Rot_A.Out.Homed_PO=0 OR Rot_B.Out.Homed_PO=0 OR Clamp_A.Out.Homed_PO=0 OR Clamp_B.Out.Homed_PO=0 THEN  
	Homed_PO:=0;
	ELSE Homed_PO:=1; END_IF
IF Mode_PI =1 THEN	
	SyncVertABSLin();
	SyncRotABS();
	SyncClampABSLin();
	msg_mode := 'Auto Mode Engaged no Jogging';
	
		// JOSEPHBARTONCHANG2-15-2023

	IF bPresetMoveTrigger THEN
		Vert_A.bPresetMoveTrigger  := TRUE;
		Rot_A.bPresetMoveTrigger   := TRUE;
		Clamp_A.bPresetMoveTrigger := TRUE;
		
		Vert_B.bPresetMoveTrigger  := TRUE;
		Rot_B.bPresetMoveTrigger   := TRUE;
		Clamp_B.bPresetMoveTrigger := TRUE;	
	
		Vert_A.bMove_PI  := TRUE;
		Rot_A.bMove_PI   := TRUE;
		Clamp_A.bMove_PI := TRUE;
		
		Vert_B.bMove_PI  := TRUE;
		Rot_B.bMove_PI   := TRUE;
		Clamp_B.bMove_PI := TRUE;
	END_IF
END_IF


IF Mode_PI =2 THEN
	SuperMode(); 
	Syncvertjog();
	SyncRotJog();
	IF ReSync_VI THEN
		
		//ReSync();
		//ReSyncFollow();
	END_IF
	msg_mode := 'Manual Mode Engaged no Auto';
END_IF
//ready to receive move command
Reset();	//just turns button on and off currently
//move to request if above is met
IF InSync() = FALSE THEN
	IF JogSeparate_VI =FALSE THEN	//if superjog mode is not enabled stop all moves if out of sync
		
	synctestbit :=1;
	//Vert_A.CancelMove(); JOSEPHBARTONCHANGE I HAVE TO PUT THIS BACK.
	//Vert_B.CancelMove();
	//Clamp_A.CancelMove();
	//Clamp_B.CancelMove();
	//Rot_A.CancelMove(); JOSEPHBARTONCHANGE Once the clamps are in synch, then i can uncomment these lines.
	//Rot_B.CancelMove();
	msg := 'Not in Sync, Move Canceled, Reset and retry home';
	ELSE
		msg := ' SuperJog Mode in Progress, Caution';
	END_IF
END_IF

METHOD PRIVATE InSync : BOOL
VAR_INPUT
END_VAR

IF Homed_PO THEN
	IF ABS(Vert_A.Out.DistancePos_PO - Vert_B.Out.DistancePos_PO) <= VertSyncTolerance_CI AND 
	ABS(Clamp_A.Out.DistancePos_PO - Clamp_B.Out.DistancePos_PO) <= VertSyncTolerance_CI  AND
  ((ABS(Rot_A.Out.DistancePos_PO - Rot_B.Out.DistancePos_PO) <= RotSyncTolerance_CI) OR bFollowerIdleDisengage) THEN
		InSync := TRUE;
	ELSE 
		InSync := TRUE; //:= FALSE; JOSEPHBARTONCHANGE3-24-2023 Change this back when needed.
		ErrorMsg_VO := 'A and B are not in Sync, check A or B for encoder slippage.';
		//IF ABS(Vert_A.Out.DistancePos_PO - Vert_B.Out.DistancePos_PO) >= VertSyncTolerance_CI THEN
		//	SyncVertMsg_VO := 'Vert: A and B not inSync'; Else SyncVertMsg_VO:='';
		//END_IF
		//IF ABS(Clamp_A.Out.DistancePos_PO - Clamp_B.Out.DistancePos_PO) >= VertSyncTolerance_CI THEN JOSEPHBARTONCHANGE
		//	SyncClampMsg_VO := 'Clamp: A and B not inSync'; ELSE SyncClampMsg_VO:='';
		//END_IF
		//IF ABS(Rot_A.Out.DistancePos_PO - Rot_B.Out.DistancePos_PO) >= RotSyncTolerance_CI THEN
		//	SyncRotMsg_VO := 'Rot: A and B not inSync'; ELSE SyncRotMsg_VO:= '';
		//END_IF
	END_IF

END_IF
END_METHOD

METHOD Reset : BOOL
VAR_INPUT
END_VAR

IF Reset_Vi = TRUE THEN
	Reset_Vi := FALSE; 
	bMoveVert_PI:=0;
	bMoveRot_PI:=0;
	bMoveClamp_PI:=0;
	SyncVertCase :=0;
	SyncRotCase :=0;
	SyncClampCase :=0;
END_IF
END_METHOD

METHOD ReSync : BOOL
VAR_INPUT
	
END_VAR
IF Homed_PO  THEN
	if Resync_VI then Resync_PI:=1; end_if
	IF ABS(Vert_A.Out.DistancePos_PO - Vert_B.Out.DistancePos_PO) <= VertSyncTolerance_CI AND 
	   ABS(Clamp_A.Out.DistancePos_PO - Clamp_B.Out.DistancePos_PO) <= VertSyncTolerance_CI THEN
		//insync is true
		//message no resync is necessary
		//when resynced reset ReSync_PI Var
		ReSync_PI :=0;
	ELSE 
		//insync is false
		//check for resync
		IF ReSync_PI THEN
			//resync requested
			JogSeparate_VI := TRUE;
			//check for part present?
			//Find A and Find B which is bigger
			IF Vert_A.Out.DistancePos_PO > Vert_B.Out.DistancePos_PO THEN
				
				CW_VI := 1;
				JogVertBExecute_VI := TRUE;
				
	
			ELSIF Vert_B.Out.DistancePos_PO > Vert_A.Out.DistancePos_PO THEN
				
				CW_VI := 0;
				JogVertBExecute_VI := TRUE;
				
			ELSE
					ReSync_PI := 0;
				
			END_IF
			
			//move the biggest down 1 pulse and move the smallest up 1 until equal
		ELSE
			JogVertBExecute_VI := FALSE;
			JogSeparate_VI := FALSE;
			
		END_IF
		
		ErrorMsg_VO := 'A and B are not in Sync, check A or B for encoder slippage.';
	END_IF
	//get closer on resync
	IF ABS(Vert_A.Out.DistancePos_PO - Vert_B.Out.DistancePos_PO) <= 2 AND ABS(Clamp_A.Out.DistancePos_PO - Clamp_B.Out.DistancePos_PO) <= 2 THEN
		//in sync
	ELSE 
		//insync is false
		//check for resync
		IF ReSync_PI THEN
			//resync requested
			//check for part present?
			//Find A and Find B which is bigger
			//will need a bmove execute button
			IF Vert_A.Out.DistancePos_PO > Vert_B.Out.DistancePos_PO THEN
				Vert_A.DistancePosReq_PI :=(Vert_A.Out.DistancePos_PO-1);
				Vert_B.DistancePosReq_PI :=(Vert_B.Out.DistancePos_PO+1);
			END_IF
			IF Vert_B.Out.DistancePos_PO > Vert_A.Out.DistancePos_PO THEN
				Vert_A.DistancePosReq_PI :=(Vert_A.Out.DistancePos_PO+1);
				Vert_B.DistancePosReq_PI :=(Vert_B.Out.DistancePos_PO-1);
			END_IF
			
			//move the biggest down 1 pulse and move the smallest up 1 until equal
			
		END_IF
		
		ErrorMsg_VO := 'A and B are not in Sync, check A or B for encoder slippage.';
	END_IF
	
	ReSync_VI := 0;
END_IF
END_METHOD

METHOD ReSyncFollow : BOOL
VAR_INPUT
END_VAR
IF Homed_PO THEN
	IF Resync_VI THEN 
		Resync_PI:=1;
	ELSIF GVL_HMI.MCR THEN
		Resync_PI:=0;
		Resync_VI:=0;
	END_IF
	
	IF ABS(Rot_A.Out.DistancePos_PO - Rot_B.Out.DistancePos_PO) <= RotSyncTolerance_CI THEN
		//insync is true
		//message no resync is necessary
		//when resynced reset ReSync_PI Var
		ReSync_PI :=0;
	ELSE 
		IF ReSync_PI THEN
			//resync requested
			//check for part present?
			//Find A and Find B which is bigger
			IF Rot_A.Out.DistancePos_PO > Rot_B.Out.DistancePos_PO THEN
				Rot_A.DistancePosReq_PI :=(Rot_A.Out.DistancePos_PO-1);
				Rot_B.DistancePosReq_PI :=(Rot_B.Out.DistancePos_PO+1);
				bMoveRot_PI :=TRUE;
				

			ELSIF Rot_B.Out.DistancePos_PO > Rot_A.Out.DistancePos_PO THEN
				Rot_A.DistancePosReq_PI := (Rot_A.Out.DistancePos_PO+1);
				Rot_B.DistancePosReq_PI := (Rot_B.Out.DistancePos_PO-1);
				bMoveRot_PI :=TRUE;
			
			ELSE
				JogRotAExecute_VI :=FALSE;
				JogRotBExecute_VI :=FALSE;
				ReSync_PI:=0;
			END_IF
			
			//move the biggest down 1 pulse and move the smallest up 1 until equal
			
		END_IF
		
		ErrorMsg_VO := 'A and B are not in Sync, check A or B for encoder slippage.';
	END_IF
	















//get closer on resync
	IF ABS(Rot_A.Out.DistancePos_PO - Rot_B.Out.DistancePos_PO) <= 2 THEN
		//in sync
	ELSE 
		//insync is false
		//check for resync
		IF ReSync_PI THEN
			//resync requested
			//check for part present?
			//Find A and Find B which is bigger
			//will need a bmove execute button
			IF Rot_A.Out.DistancePos_PO > Rot_B.Out.DistancePos_PO THEN
				Rot_A.DistancePosReq_PI :=(Rot_A.Out.DistancePos_PO-1);
				Rot_B.DistancePosReq_PI :=(Rot_B.Out.DistancePos_PO+1);
			END_IF
			IF Rot_B.Out.DistancePos_PO > Rot_A.Out.DistancePos_PO THEN
				Rot_A.DistancePosReq_PI :=(Rot_A.Out.DistancePos_PO+1);
				Rot_B.DistancePosReq_PI :=(Rot_B.Out.DistancePos_PO-1);
			END_IF
			
			//move the biggest down 1 pulse and move the smallest up 1 until equal
			
		END_IF
		
		ErrorMsg_VO := 'A and B are not in Sync, check A or B for encoder slippage.';
	END_IF
	
	
END_IF
END_METHOD

